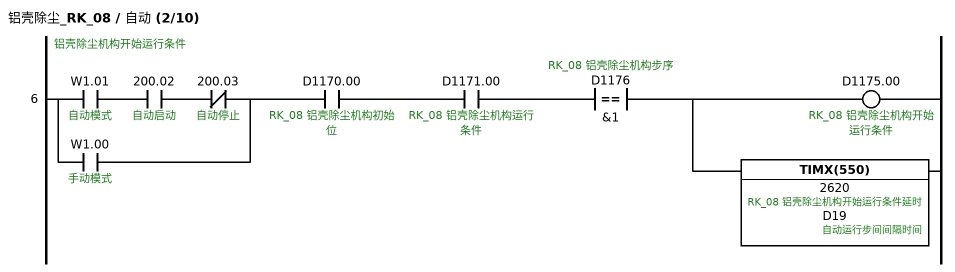
; [picture p624: 铝壳除尘_RK_08 / 自动, rungs 6-6]
; rung 6: 铝壳除尘机构开始运行条件
LD W1.01  ; 自动模式
AND 200.02  ; 自动启动
ANDNOT 200.03  ; 自动停止
OR W1.00  ; 手动模式
AND D1170.00  ; RK_08 铝壳除尘机构初始位
AND D1171.00  ; RK_08 铝壳除尘机构运行条件
AND=(300) D1176 &1  ; RK_08 铝壳除尘机构步序
OUT D1175.00  ; RK_08 铝壳除尘机构开始运行条件
TIMX(550) 2620 D19  ; 自动运行步间间隔时间, RK_08 铝壳除尘机构开始运行条件延时

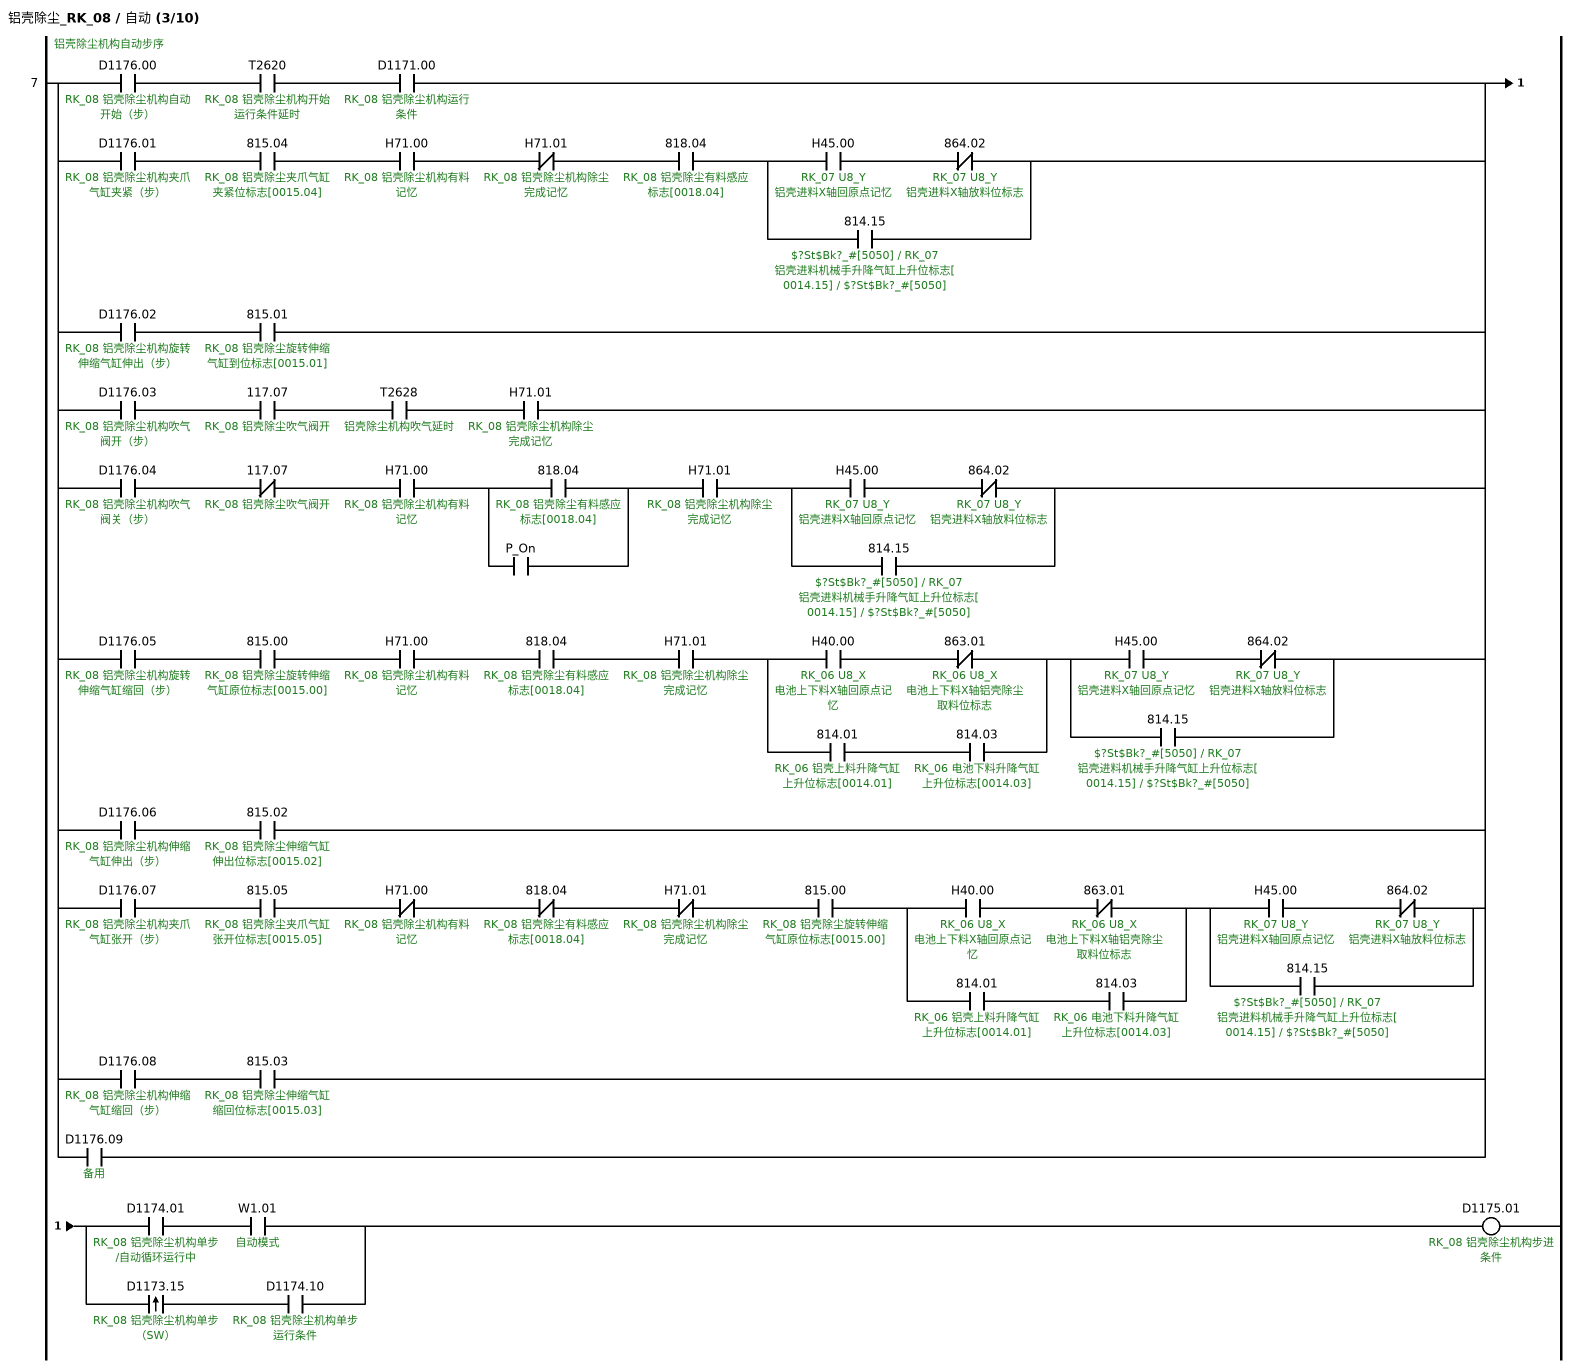
; rung 7: 铝壳除尘机构自动步序
LD D1176.00  ; RK_08 铝壳除尘机构自动开始（步）
AND T2620  ; RK_08 铝壳除尘机构开始运行条件延时
AND D1171.00  ; RK_08 铝壳除尘机构运行条件
LD D1176.01  ; RK_08 铝壳除尘机构夹爪气缸夹紧（步）
AND 815.04  ; RK_08 铝壳除尘夹爪气缸夹紧位标志[0015.04]
AND H71.00  ; RK_08 铝壳除尘机构有料记忆
ANDNOT H71.01  ; RK_08 铝壳除尘机构除尘完成记忆
AND 818.04  ; RK_08 铝壳除尘有料感应标志[0018.04]
LD H45.00  ; RK_07 U8_Y 铝壳进料X轴回原点记忆
ANDNOT 864.02  ; RK_07 U8_Y 铝壳进料X轴放料位标志
OR 814.15  ; $?St$Bk?_#[5050] / RK_07 铝壳进料机械手升降气缸上升位标志[0014.15] / $?St$Bk?_#[5050]
ANDLD
ORLD
LD D1176.02  ; RK_08 铝壳除尘机构旋转伸缩气缸伸出（步）
AND 815.01  ; RK_08 铝壳除尘旋转伸缩气缸到位标志[0015.01]
ORLD
LD D1176.03  ; RK_08 铝壳除尘机构吹气阀开（步）
AND 117.07  ; RK_08 铝壳除尘吹气阀开
AND T2628  ; 铝壳除尘机构吹气延时
AND H71.01  ; RK_08 铝壳除尘机构除尘完成记忆
ORLD
LD D1176.04  ; RK_08 铝壳除尘机构吹气阀关（步）
ANDNOT 117.07  ; RK_08 铝壳除尘吹气阀开
AND H71.00  ; RK_08 铝壳除尘机构有料记忆
LD 818.04  ; RK_08 铝壳除尘有料感应标志[0018.04]
OR P_On
ANDLD
AND H71.01  ; RK_08 铝壳除尘机构除尘完成记忆
LD H45.00  ; RK_07 U8_Y 铝壳进料X轴回原点记忆
ANDNOT 864.02  ; RK_07 U8_Y 铝壳进料X轴放料位标志
OR 814.15  ; $?St$Bk?_#[5050] / RK_07 铝壳进料机械手升降气缸上升位标志[0014.15] / $?St$Bk?_#[5050]
ANDLD
ORLD
LD D1176.05  ; RK_08 铝壳除尘机构旋转伸缩气缸缩回（步）
AND 815.00  ; RK_08 铝壳除尘旋转伸缩气缸原位标志[0015.00]
AND H71.00  ; RK_08 铝壳除尘机构有料记忆
AND 818.04  ; RK_08 铝壳除尘有料感应标志[0018.04]
AND H71.01  ; RK_08 铝壳除尘机构除尘完成记忆
LD H40.00  ; RK_06 U8_X 电池上下料X轴回原点记忆
ANDNOT 863.01  ; RK_06 U8_X 电池上下料X轴铝壳除尘取料位标志
LD 814.01  ; RK_06 铝壳上料升降气缸上升位标志[0014.01]
AND 814.03  ; RK_06 电池下料升降气缸上升位标志[0014.03]
ORLD
ANDLD
LD H45.00  ; RK_07 U8_Y 铝壳进料X轴回原点记忆
ANDNOT 864.02  ; RK_07 U8_Y 铝壳进料X轴放料位标志
OR 814.15  ; $?St$Bk?_#[5050] / RK_07 铝壳进料机械手升降气缸上升位标志[0014.15] / $?St$Bk?_#[5050]
ANDLD
ORLD
LD D1176.06  ; RK_08 铝壳除尘机构伸缩气缸伸出（步）
AND 815.02  ; RK_08 铝壳除尘伸缩气缸伸出位标志[0015.02]
ORLD
LD D1176.07  ; RK_08 铝壳除尘机构夹爪气缸张开（步）
AND 815.05  ; RK_08 铝壳除尘夹爪气缸张开位标志[0015.05]
ANDNOT H71.00  ; RK_08 铝壳除尘机构有料记忆
ANDNOT 818.04  ; RK_08 铝壳除尘有料感应标志[0018.04]
ANDNOT H71.01  ; RK_08 铝壳除尘机构除尘完成记忆
AND 815.00  ; RK_08 铝壳除尘旋转伸缩气缸原位标志[0015.00]
LD H40.00  ; RK_06 U8_X 电池上下料X轴回原点记忆
ANDNOT 863.01  ; RK_06 U8_X 电池上下料X轴铝壳除尘取料位标志
LD 814.01  ; RK_06 铝壳上料升降气缸上升位标志[0014.01]
AND 814.03  ; RK_06 电池下料升降气缸上升位标志[0014.03]
ORLD
ANDLD
LD H45.00  ; RK_07 U8_Y 铝壳进料X轴回原点记忆
ANDNOT 864.02  ; RK_07 U8_Y 铝壳进料X轴放料位标志
OR 814.15  ; $?St$Bk?_#[5050] / RK_07 铝壳进料机械手升降气缸上升位标志[0014.15] / $?St$Bk?_#[5050]
ANDLD
ORLD
LD D1176.08  ; RK_08 铝壳除尘机构伸缩气缸缩回（步）
AND 815.03  ; RK_08 铝壳除尘伸缩气缸缩回位标志[0015.03]
ORLD
OR D1176.09  ; 备用
LD D1174.01  ; RK_08 铝壳除尘机构单步/自动循环运行中
AND W1.01  ; 自动模式
@LD D1173.15  ; RK_08 铝壳除尘机构单步（SW）
AND D1174.10  ; RK_08 铝壳除尘机构单步运行条件
ORLD
ANDLD
OUT D1175.01  ; RK_08 铝壳除尘机构步进条件

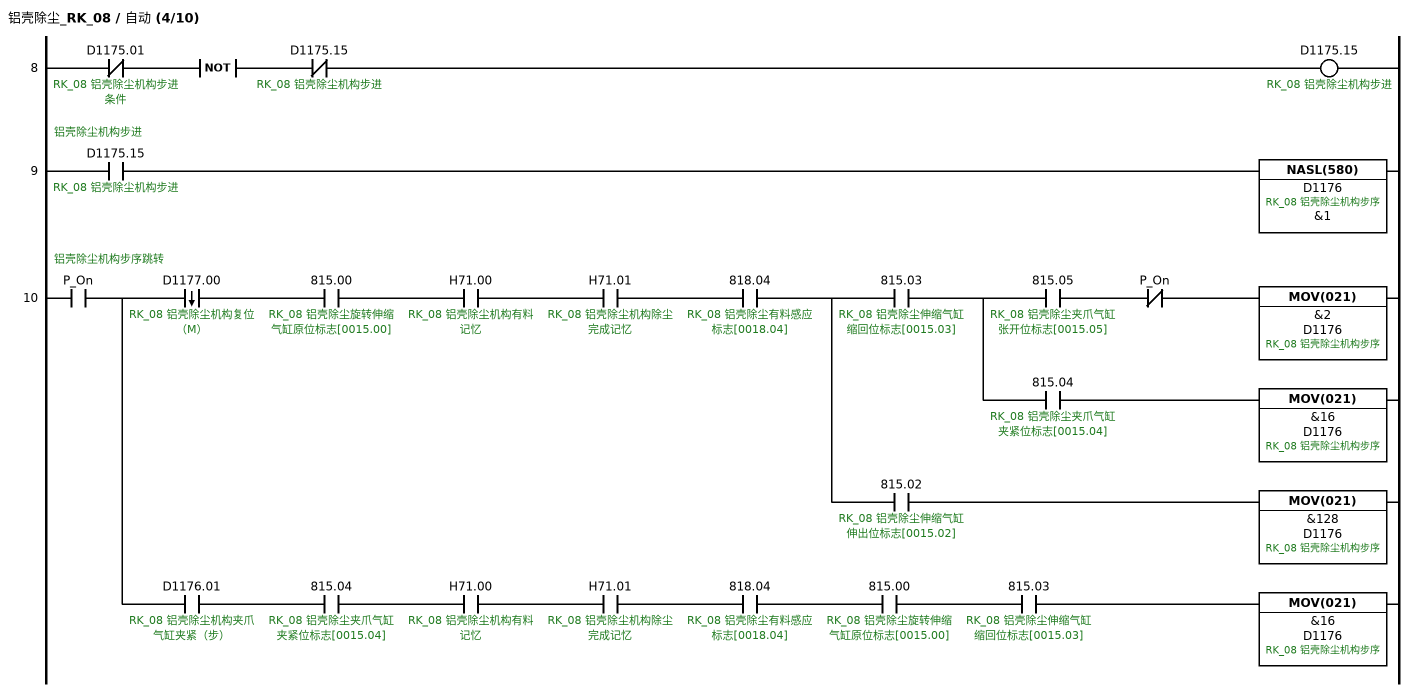
; rung 8
LDNOT D1175.01  ; RK_08 铝壳除尘机构步进条件
NOT(520)
ANDNOT D1175.15  ; RK_08 铝壳除尘机构步进
OUT D1175.15  ; RK_08 铝壳除尘机构步进
; rung 9: 铝壳除尘机构步进
LD D1175.15  ; RK_08 铝壳除尘机构步进
NASL(580) D1176 &1  ; RK_08 铝壳除尘机构步序
; rung 10: 铝壳除尘机构步序跳转
LD P_On
OUT TR0
%AND D1177.00  ; RK_08 铝壳除尘机构复位（M）
AND 815.00  ; RK_08 铝壳除尘旋转伸缩气缸原位标志[0015.00]
AND H71.00  ; RK_08 铝壳除尘机构有料记忆
AND H71.01  ; RK_08 铝壳除尘机构除尘完成记忆
AND 818.04  ; RK_08 铝壳除尘有料感应标志[0018.04]
OUT TR1
AND 815.03  ; RK_08 铝壳除尘伸缩气缸缩回位标志[0015.03]
OUT TR2
AND 815.05  ; RK_08 铝壳除尘夹爪气缸张开位标志[0015.05]
ANDNOT P_On
MOV(021) &2 D1176  ; RK_08 铝壳除尘机构步序  // RK_08 铝壳除尘机构夹爪气缸夹紧步（D1176.01）
LD TR2
AND 815.04  ; RK_08 铝壳除尘夹爪气缸夹紧位标志[0015.04]
MOV(021) &16 D1176  ; RK_08 铝壳除尘机构步序  // RK_08 铝壳除尘机构吹气阀关步（D1176.04）
LD TR1
AND 815.02  ; RK_08 铝壳除尘伸缩气缸伸出位标志[0015.02]
MOV(021) &128 D1176  ; RK_08 铝壳除尘机构步序  // RK_08 铝壳除尘机构夹爪气缸张开步（D1176.07）
LD TR0
AND D1176.01  ; RK_08 铝壳除尘机构夹爪气缸夹紧（步）
AND 815.04  ; RK_08 铝壳除尘夹爪气缸夹紧位标志[0015.04]
AND H71.00  ; RK_08 铝壳除尘机构有料记忆
AND H71.01  ; RK_08 铝壳除尘机构除尘完成记忆
AND 818.04  ; RK_08 铝壳除尘有料感应标志[0018.04]
AND 815.00  ; RK_08 铝壳除尘旋转伸缩气缸原位标志[0015.00]
AND 815.03  ; RK_08 铝壳除尘伸缩气缸缩回位标志[0015.03]
MOV(021) &16 D1176  ; RK_08 铝壳除尘机构步序  // RK_08 铝壳除尘机构吹气阀关步（D1176.04）

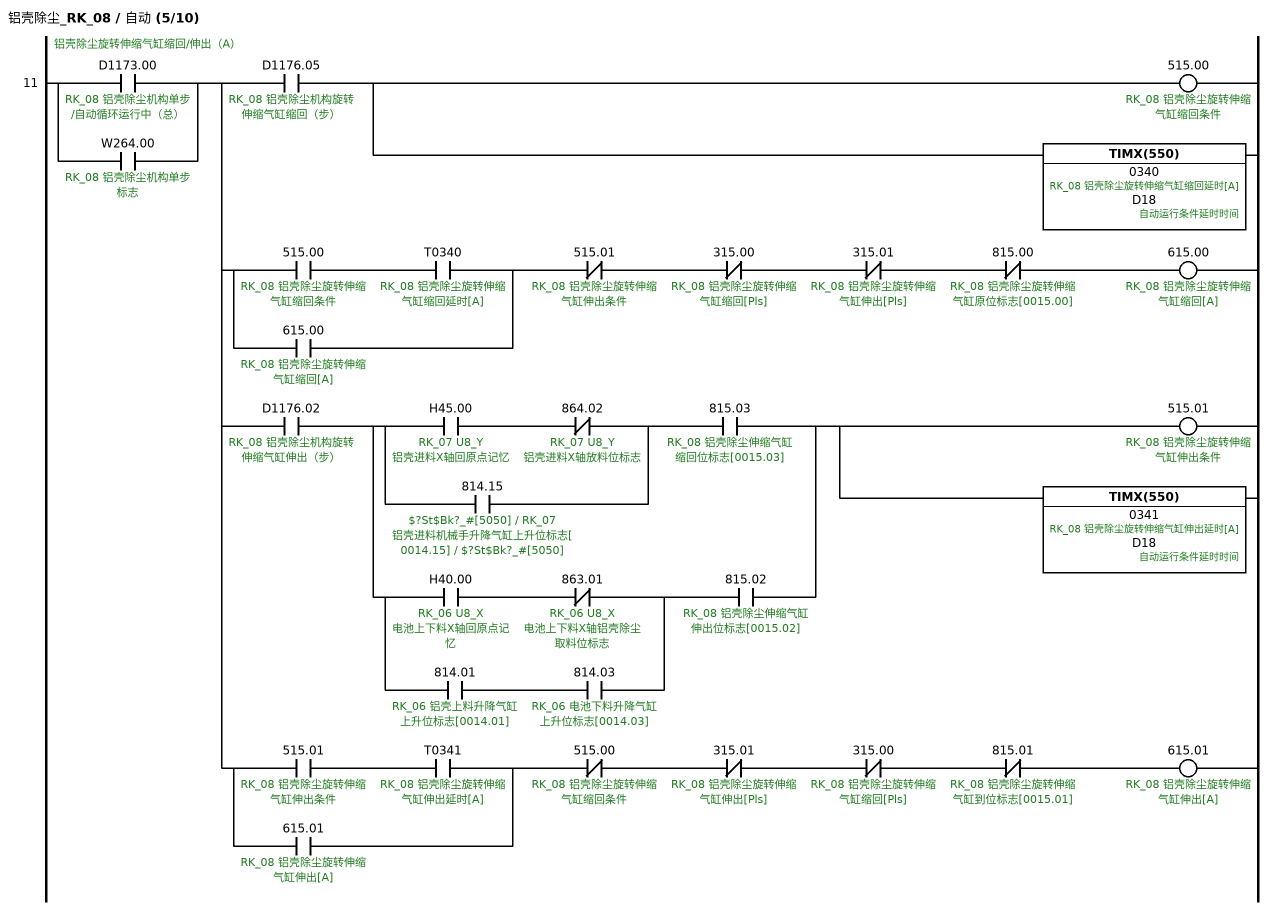
; rung 11: 铝壳除尘旋转伸缩气缸缩回/伸出（A）
LD D1173.00  ; RK_08 铝壳除尘机构单步/自动循环运行中（总）
OR W264.00  ; RK_08 铝壳除尘机构单步标志
OUT TR0
AND D1176.05  ; RK_08 铝壳除尘机构旋转伸缩气缸缩回（步）
OUT 515.00  ; RK_08 铝壳除尘旋转伸缩气缸缩回条件
TIMX(550) 0340 D18  ; 自动运行条件延时时间, RK_08 铝壳除尘旋转伸缩气缸缩回延时[A]
LD TR0
LD 515.00  ; RK_08 铝壳除尘旋转伸缩气缸缩回条件
AND T0340  ; RK_08 铝壳除尘旋转伸缩气缸缩回延时[A]
OR 615.00  ; RK_08 铝壳除尘旋转伸缩气缸缩回[A]
ANDLD
ANDNOT 515.01  ; RK_08 铝壳除尘旋转伸缩气缸伸出条件
ANDNOT 315.00  ; RK_08 铝壳除尘旋转伸缩气缸缩回[Pls]
ANDNOT 315.01  ; RK_08 铝壳除尘旋转伸缩气缸伸出[Pls]
ANDNOT 815.00  ; RK_08 铝壳除尘旋转伸缩气缸原位标志[0015.00]
OUT 615.00  ; RK_08 铝壳除尘旋转伸缩气缸缩回[A]
LD TR0
AND D1176.02  ; RK_08 铝壳除尘机构旋转伸缩气缸伸出（步）
LD H45.00  ; RK_07 U8_Y 铝壳进料X轴回原点记忆
ANDNOT 864.02  ; RK_07 U8_Y 铝壳进料X轴放料位标志
OR 814.15  ; $?St$Bk?_#[5050] / RK_07 铝壳进料机械手升降气缸上升位标志[0014.15] / $?St$Bk?_#[5050]
AND 815.03  ; RK_08 铝壳除尘伸缩气缸缩回位标志[0015.03]
LD H40.00  ; RK_06 U8_X 电池上下料X轴回原点记忆
ANDNOT 863.01  ; RK_06 U8_X 电池上下料X轴铝壳除尘取料位标志
LD 814.01  ; RK_06 铝壳上料升降气缸上升位标志[0014.01]
AND 814.03  ; RK_06 电池下料升降气缸上升位标志[0014.03]
ORLD
AND 815.02  ; RK_08 铝壳除尘伸缩气缸伸出位标志[0015.02]
ORLD
ANDLD
OUT 515.01  ; RK_08 铝壳除尘旋转伸缩气缸伸出条件
TIMX(550) 0341 D18  ; 自动运行条件延时时间, RK_08 铝壳除尘旋转伸缩气缸伸出延时[A]
LD TR0
LD 515.01  ; RK_08 铝壳除尘旋转伸缩气缸伸出条件
AND T0341  ; RK_08 铝壳除尘旋转伸缩气缸伸出延时[A]
OR 615.01  ; RK_08 铝壳除尘旋转伸缩气缸伸出[A]
ANDLD
ANDNOT 515.00  ; RK_08 铝壳除尘旋转伸缩气缸缩回条件
ANDNOT 315.01  ; RK_08 铝壳除尘旋转伸缩气缸伸出[Pls]
ANDNOT 315.00  ; RK_08 铝壳除尘旋转伸缩气缸缩回[Pls]
ANDNOT 815.01  ; RK_08 铝壳除尘旋转伸缩气缸到位标志[0015.01]
OUT 615.01  ; RK_08 铝壳除尘旋转伸缩气缸伸出[A]

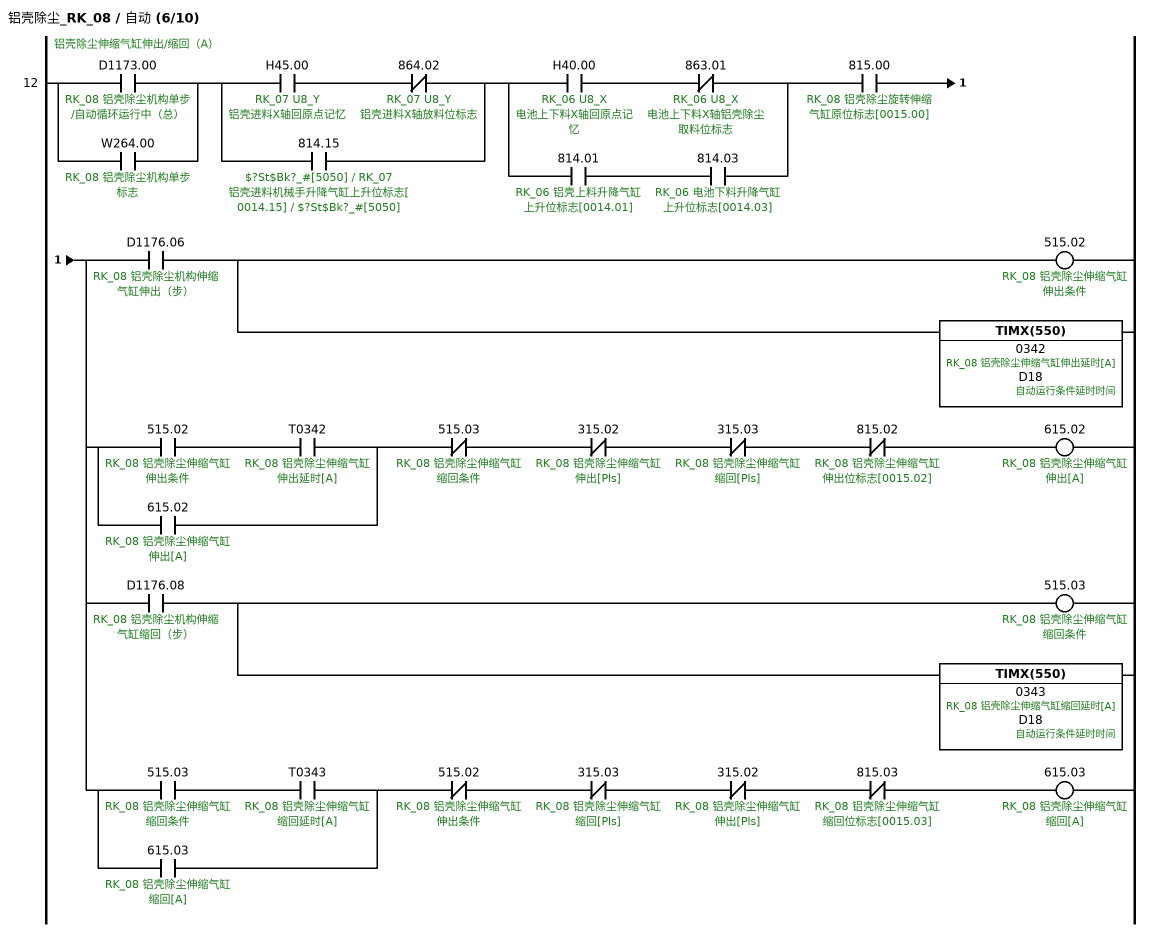
; rung 12: 铝壳除尘伸缩气缸伸出/缩回（A）
LD D1173.00  ; RK_08 铝壳除尘机构单步/自动循环运行中（总）
OR W264.00  ; RK_08 铝壳除尘机构单步标志
LD H45.00  ; RK_07 U8_Y 铝壳进料X轴回原点记忆
ANDNOT 864.02  ; RK_07 U8_Y 铝壳进料X轴放料位标志
OR 814.15  ; $?St$Bk?_#[5050] / RK_07 铝壳进料机械手升降气缸上升位标志[0014.15] / $?St$Bk?_#[5050]
ANDLD
LD H40.00  ; RK_06 U8_X 电池上下料X轴回原点记忆
ANDNOT 863.01  ; RK_06 U8_X 电池上下料X轴铝壳除尘取料位标志
LD 814.01  ; RK_06 铝壳上料升降气缸上升位标志[0014.01]
AND 814.03  ; RK_06 电池下料升降气缸上升位标志[0014.03]
ORLD
ANDLD
AND 815.00  ; RK_08 铝壳除尘旋转伸缩气缸原位标志[0015.00]
OUT TR0
AND D1176.06  ; RK_08 铝壳除尘机构伸缩气缸伸出（步）
OUT 515.02  ; RK_08 铝壳除尘伸缩气缸伸出条件
TIMX(550) 0342 D18  ; 自动运行条件延时时间, RK_08 铝壳除尘伸缩气缸伸出延时[A]
LD TR0
LD 515.02  ; RK_08 铝壳除尘伸缩气缸伸出条件
AND T0342  ; RK_08 铝壳除尘伸缩气缸伸出延时[A]
OR 615.02  ; RK_08 铝壳除尘伸缩气缸伸出[A]
ANDLD
ANDNOT 515.03  ; RK_08 铝壳除尘伸缩气缸缩回条件
ANDNOT 315.02  ; RK_08 铝壳除尘伸缩气缸伸出[Pls]
ANDNOT 315.03  ; RK_08 铝壳除尘伸缩气缸缩回[Pls]
ANDNOT 815.02  ; RK_08 铝壳除尘伸缩气缸伸出位标志[0015.02]
OUT 615.02  ; RK_08 铝壳除尘伸缩气缸伸出[A]
LD TR0
AND D1176.08  ; RK_08 铝壳除尘机构伸缩气缸缩回（步）
OUT 515.03  ; RK_08 铝壳除尘伸缩气缸缩回条件
TIMX(550) 0343 D18  ; 自动运行条件延时时间, RK_08 铝壳除尘伸缩气缸缩回延时[A]
LD TR0
LD 515.03  ; RK_08 铝壳除尘伸缩气缸缩回条件
AND T0343  ; RK_08 铝壳除尘伸缩气缸缩回延时[A]
OR 615.03  ; RK_08 铝壳除尘伸缩气缸缩回[A]
ANDLD
ANDNOT 515.02  ; RK_08 铝壳除尘伸缩气缸伸出条件
ANDNOT 315.03  ; RK_08 铝壳除尘伸缩气缸缩回[Pls]
ANDNOT 315.02  ; RK_08 铝壳除尘伸缩气缸伸出[Pls]
ANDNOT 815.03  ; RK_08 铝壳除尘伸缩气缸缩回位标志[0015.03]
OUT 615.03  ; RK_08 铝壳除尘伸缩气缸缩回[A]

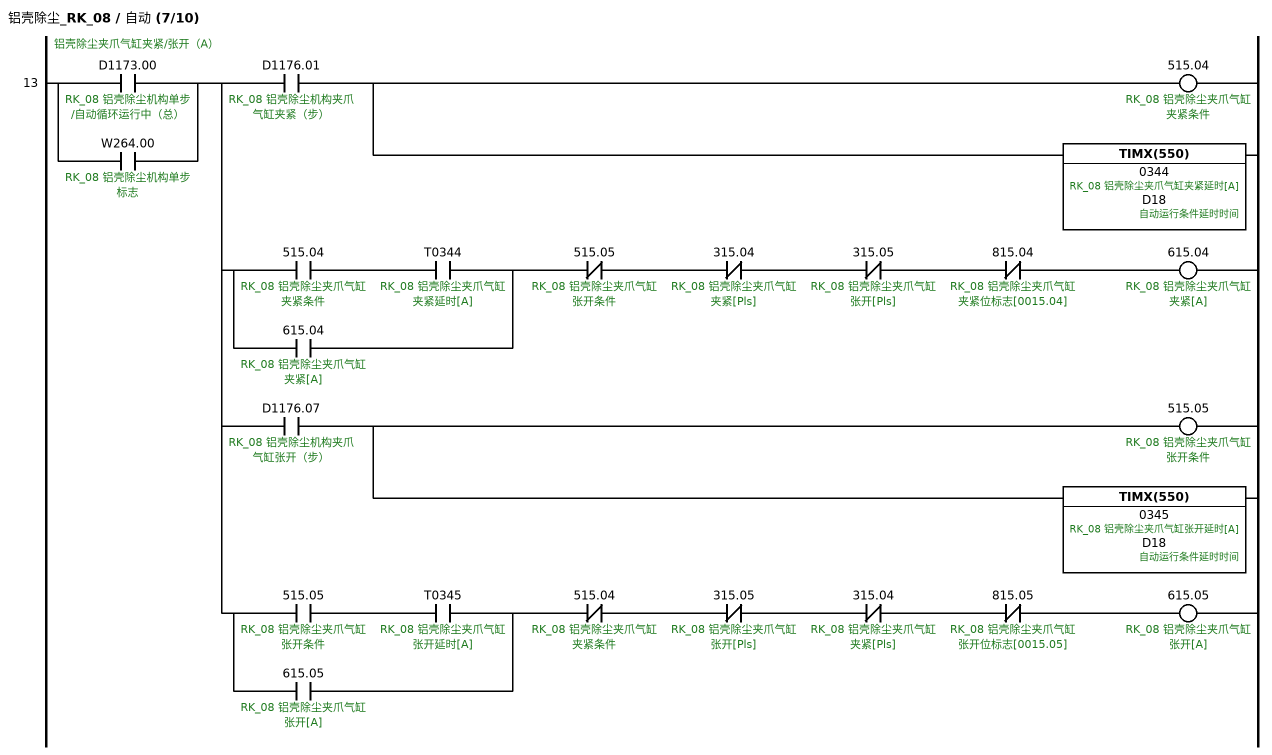
; rung 13: 铝壳除尘夹爪气缸夹紧/张开（A）
LD D1173.00  ; RK_08 铝壳除尘机构单步/自动循环运行中（总）
OR W264.00  ; RK_08 铝壳除尘机构单步标志
OUT TR0
AND D1176.01  ; RK_08 铝壳除尘机构夹爪气缸夹紧（步）
OUT 515.04  ; RK_08 铝壳除尘夹爪气缸夹紧条件
TIMX(550) 0344 D18  ; 自动运行条件延时时间, RK_08 铝壳除尘夹爪气缸夹紧延时[A]
LD TR0
LD 515.04  ; RK_08 铝壳除尘夹爪气缸夹紧条件
AND T0344  ; RK_08 铝壳除尘夹爪气缸夹紧延时[A]
OR 615.04  ; RK_08 铝壳除尘夹爪气缸夹紧[A]
ANDLD
ANDNOT 515.05  ; RK_08 铝壳除尘夹爪气缸张开条件
ANDNOT 315.04  ; RK_08 铝壳除尘夹爪气缸夹紧[Pls]
ANDNOT 315.05  ; RK_08 铝壳除尘夹爪气缸张开[Pls]
ANDNOT 815.04  ; RK_08 铝壳除尘夹爪气缸夹紧位标志[0015.04]
OUT 615.04  ; RK_08 铝壳除尘夹爪气缸夹紧[A]
LD TR0
AND D1176.07  ; RK_08 铝壳除尘机构夹爪气缸张开（步）
OUT 515.05  ; RK_08 铝壳除尘夹爪气缸张开条件
TIMX(550) 0345 D18  ; 自动运行条件延时时间, RK_08 铝壳除尘夹爪气缸张开延时[A]
LD TR0
LD 515.05  ; RK_08 铝壳除尘夹爪气缸张开条件
AND T0345  ; RK_08 铝壳除尘夹爪气缸张开延时[A]
OR 615.05  ; RK_08 铝壳除尘夹爪气缸张开[A]
ANDLD
ANDNOT 515.04  ; RK_08 铝壳除尘夹爪气缸夹紧条件
ANDNOT 315.05  ; RK_08 铝壳除尘夹爪气缸张开[Pls]
ANDNOT 315.04  ; RK_08 铝壳除尘夹爪气缸夹紧[Pls]
ANDNOT 815.05  ; RK_08 铝壳除尘夹爪气缸张开位标志[0015.05]
OUT 615.05  ; RK_08 铝壳除尘夹爪气缸张开[A]

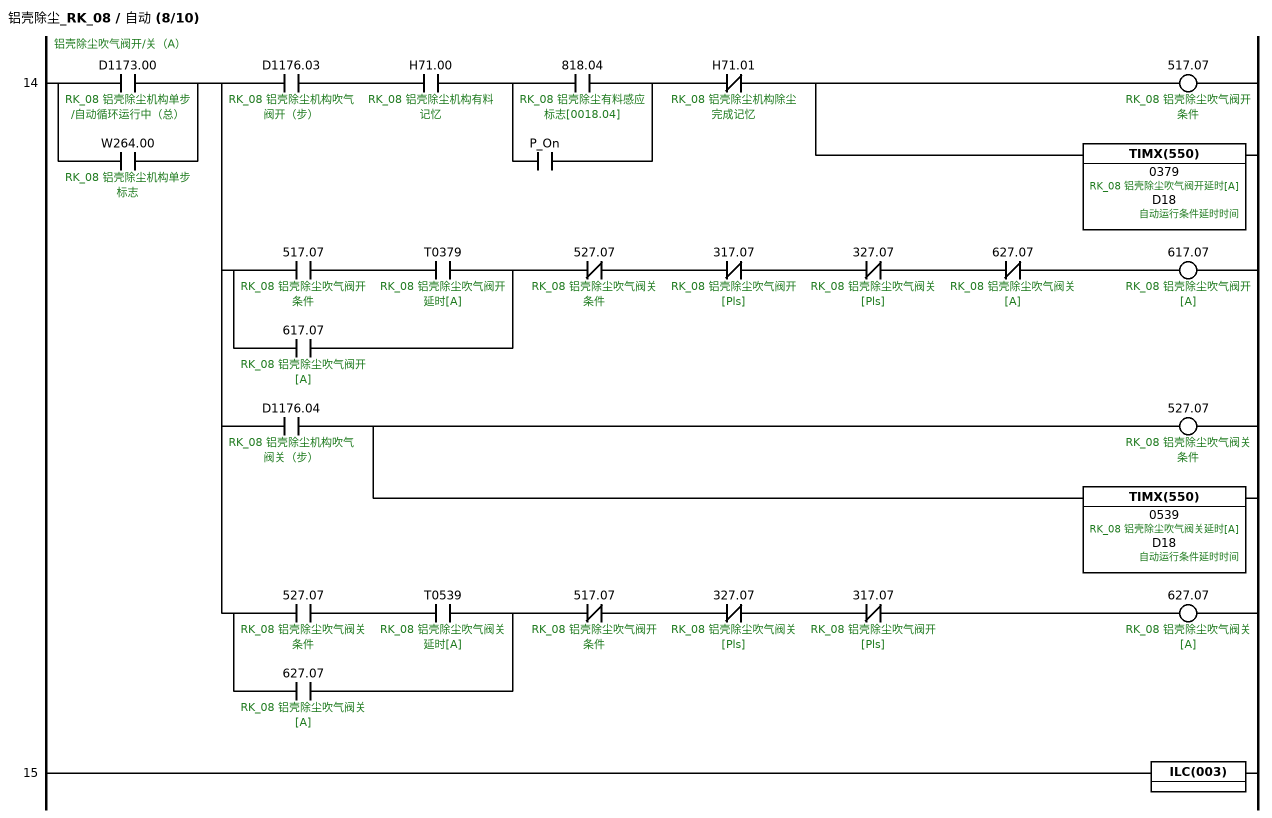
; rung 14: 铝壳除尘吹气阀开/关（A）
LD D1173.00  ; RK_08 铝壳除尘机构单步/自动循环运行中（总）
OR W264.00  ; RK_08 铝壳除尘机构单步标志
OUT TR0
AND D1176.03  ; RK_08 铝壳除尘机构吹气阀开（步）
AND H71.00  ; RK_08 铝壳除尘机构有料记忆
LD 818.04  ; RK_08 铝壳除尘有料感应标志[0018.04]
OR P_On
ANDLD
ANDNOT H71.01  ; RK_08 铝壳除尘机构除尘完成记忆
OUT 517.07  ; RK_08 铝壳除尘吹气阀开条件
TIMX(550) 0379 D18  ; 自动运行条件延时时间, RK_08 铝壳除尘吹气阀开延时[A]
LD TR0
LD 517.07  ; RK_08 铝壳除尘吹气阀开条件
AND T0379  ; RK_08 铝壳除尘吹气阀开延时[A]
OR 617.07  ; RK_08 铝壳除尘吹气阀开[A]
ANDLD
ANDNOT 527.07  ; RK_08 铝壳除尘吹气阀关条件
ANDNOT 317.07  ; RK_08 铝壳除尘吹气阀开[Pls]
ANDNOT 327.07  ; RK_08 铝壳除尘吹气阀关[Pls]
ANDNOT 627.07  ; RK_08 铝壳除尘吹气阀关[A]
OUT 617.07  ; RK_08 铝壳除尘吹气阀开[A]
LD TR0
AND D1176.04  ; RK_08 铝壳除尘机构吹气阀关（步）
OUT 527.07  ; RK_08 铝壳除尘吹气阀关条件
TIMX(550) 0539 D18  ; 自动运行条件延时时间, RK_08 铝壳除尘吹气阀关延时[A]
LD TR0
LD 527.07  ; RK_08 铝壳除尘吹气阀关条件
AND T0539  ; RK_08 铝壳除尘吹气阀关延时[A]
OR 627.07  ; RK_08 铝壳除尘吹气阀关[A]
ANDLD
ANDNOT 517.07  ; RK_08 铝壳除尘吹气阀开条件
ANDNOT 327.07  ; RK_08 铝壳除尘吹气阀关[Pls]
ANDNOT 317.07  ; RK_08 铝壳除尘吹气阀开[Pls]
OUT 627.07  ; RK_08 铝壳除尘吹气阀关[A]
; rung 15
ILC(003)

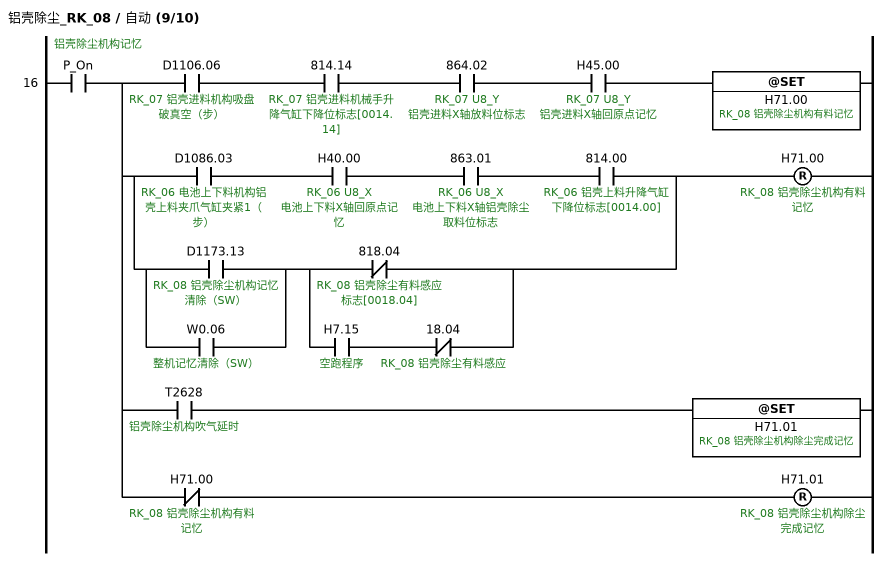
; rung 16: 铝壳除尘机构记忆
LD P_On
OUT TR0
AND D1106.06  ; RK_07 铝壳进料机构吸盘破真空（步）
AND 814.14  ; RK_07 铝壳进料机械手升降气缸下降位标志[0014.14]
AND 864.02  ; RK_07 U8_Y 铝壳进料X轴放料位标志
AND H45.00  ; RK_07 U8_Y 铝壳进料X轴回原点记忆
@SET H71.00  ; RK_08 铝壳除尘机构有料记忆
LD TR0
LD D1086.03  ; RK_06 电池上下料机构铝壳上料夹爪气缸夹紧1（步）
AND H40.00  ; RK_06 U8_X 电池上下料X轴回原点记忆
AND 863.01  ; RK_06 U8_X 电池上下料X轴铝壳除尘取料位标志
AND 814.00  ; RK_06 铝壳上料升降气缸下降位标志[0014.00]
LD D1173.13  ; RK_08 铝壳除尘机构记忆清除（SW）
OR W0.06  ; 整机记忆清除（SW）
LDNOT 818.04  ; RK_08 铝壳除尘有料感应标志[0018.04]
LD H7.15  ; 空跑程序
ANDNOT 18.04  ; RK_08 铝壳除尘有料感应
ORLD
ANDLD
ORLD
ANDLD
RSET H71.00  ; RK_08 铝壳除尘机构有料记忆
LD TR0
AND T2628  ; 铝壳除尘机构吹气延时
@SET H71.01  ; RK_08 铝壳除尘机构除尘完成记忆
LD TR0
ANDNOT H71.00  ; RK_08 铝壳除尘机构有料记忆
RSET H71.01  ; RK_08 铝壳除尘机构除尘完成记忆

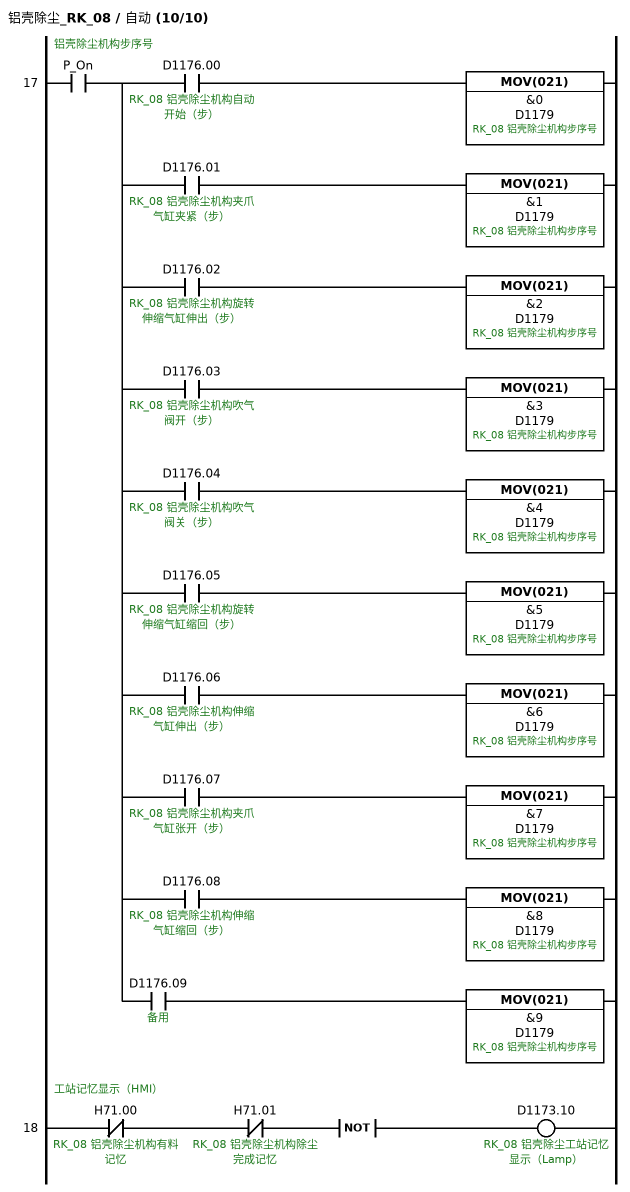
; rung 17: 铝壳除尘机构步序号
LD P_On
OUT TR0
AND D1176.00  ; RK_08 铝壳除尘机构自动开始（步）
MOV(021) &0 D1179  ; RK_08 铝壳除尘机构步序号
LD TR0
AND D1176.01  ; RK_08 铝壳除尘机构夹爪气缸夹紧（步）
MOV(021) &1 D1179  ; RK_08 铝壳除尘机构步序号
LD TR0
AND D1176.02  ; RK_08 铝壳除尘机构旋转伸缩气缸伸出（步）
MOV(021) &2 D1179  ; RK_08 铝壳除尘机构步序号
LD TR0
AND D1176.03  ; RK_08 铝壳除尘机构吹气阀开（步）
MOV(021) &3 D1179  ; RK_08 铝壳除尘机构步序号
LD TR0
AND D1176.04  ; RK_08 铝壳除尘机构吹气阀关（步）
MOV(021) &4 D1179  ; RK_08 铝壳除尘机构步序号
LD TR0
AND D1176.05  ; RK_08 铝壳除尘机构旋转伸缩气缸缩回（步）
MOV(021) &5 D1179  ; RK_08 铝壳除尘机构步序号
LD TR0
AND D1176.06  ; RK_08 铝壳除尘机构伸缩气缸伸出（步）
MOV(021) &6 D1179  ; RK_08 铝壳除尘机构步序号
LD TR0
AND D1176.07  ; RK_08 铝壳除尘机构夹爪气缸张开（步）
MOV(021) &7 D1179  ; RK_08 铝壳除尘机构步序号
LD TR0
AND D1176.08  ; RK_08 铝壳除尘机构伸缩气缸缩回（步）
MOV(021) &8 D1179  ; RK_08 铝壳除尘机构步序号
LD TR0
AND D1176.09  ; 备用
MOV(021) &9 D1179  ; RK_08 铝壳除尘机构步序号
; rung 18: 工站记忆显示（HMI）
LDNOT H71.00  ; RK_08 铝壳除尘机构有料记忆
ANDNOT H71.01  ; RK_08 铝壳除尘机构除尘完成记忆
NOT(520)
OUT D1173.10  ; RK_08 铝壳除尘工站记忆显示（Lamp）

### Section 复位

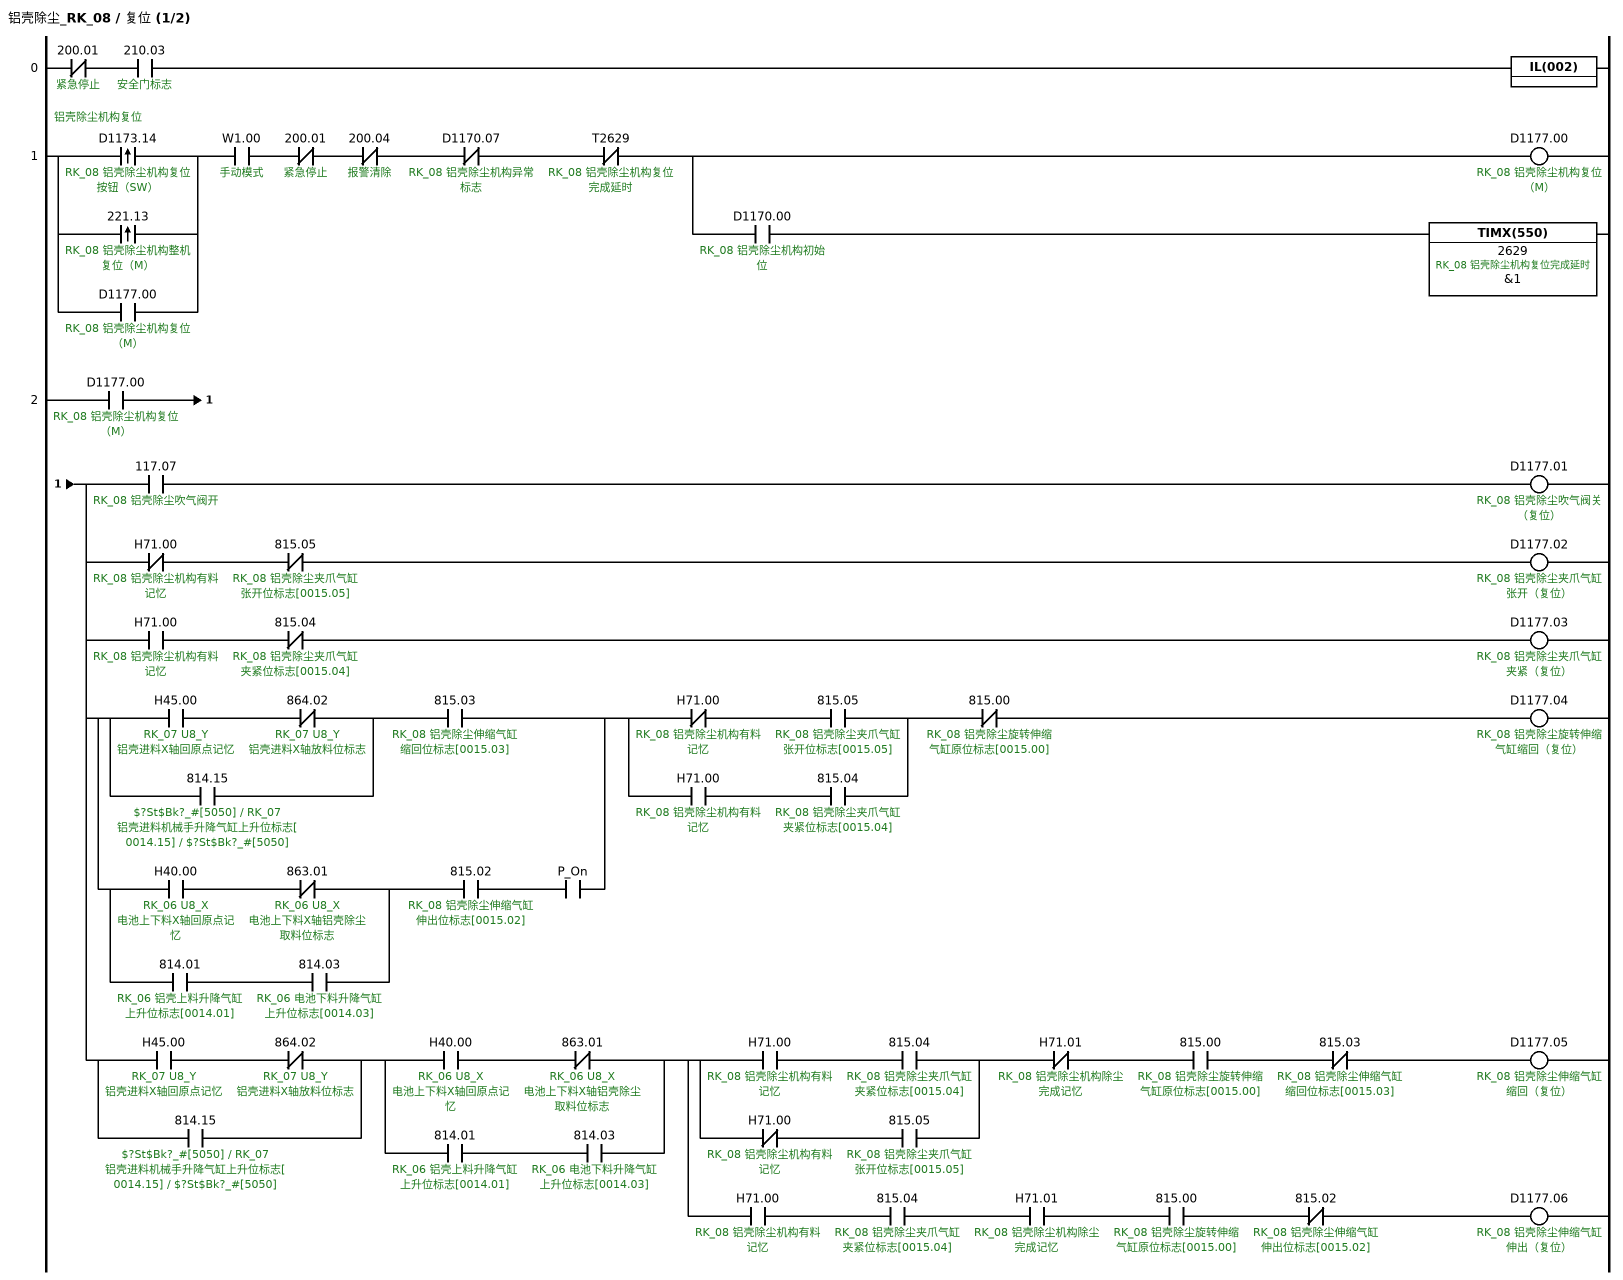
; rung 0
LDNOT 200.01  ; 紧急停止
AND 210.03  ; 安全门标志
IL(002)
; rung 1: 铝壳除尘机构复位
@LD D1173.14  ; RK_08 铝壳除尘机构复位按钮（SW）
@OR 221.13  ; RK_08 铝壳除尘机构整机复位（M）
OR D1177.00  ; RK_08 铝壳除尘机构复位（M）
AND W1.00  ; 手动模式
ANDNOT 200.01  ; 紧急停止
ANDNOT 200.04  ; 报警清除
ANDNOT D1170.07  ; RK_08 铝壳除尘机构异常标志
ANDNOT T2629  ; RK_08 铝壳除尘机构复位完成延时
OUT D1177.00  ; RK_08 铝壳除尘机构复位（M）
AND D1170.00  ; RK_08 铝壳除尘机构初始位
TIMX(550) 2629 &1  ; RK_08 铝壳除尘机构复位完成延时
; rung 2
LD D1177.00  ; RK_08 铝壳除尘机构复位（M）
OUT TR0
AND 117.07  ; RK_08 铝壳除尘吹气阀开
OUT D1177.01  ; RK_08 铝壳除尘吹气阀关（复位）
LD TR0
ANDNOT H71.00  ; RK_08 铝壳除尘机构有料记忆
ANDNOT 815.05  ; RK_08 铝壳除尘夹爪气缸张开位标志[0015.05]
OUT D1177.02  ; RK_08 铝壳除尘夹爪气缸张开（复位）
LD TR0
AND H71.00  ; RK_08 铝壳除尘机构有料记忆
ANDNOT 815.04  ; RK_08 铝壳除尘夹爪气缸夹紧位标志[0015.04]
OUT D1177.03  ; RK_08 铝壳除尘夹爪气缸夹紧（复位）
LD TR0
LD H45.00  ; RK_07 U8_Y 铝壳进料X轴回原点记忆
ANDNOT 864.02  ; RK_07 U8_Y 铝壳进料X轴放料位标志
OR 814.15  ; $?St$Bk?_#[5050] / RK_07 铝壳进料机械手升降气缸上升位标志[0014.15] / $?St$Bk?_#[5050]
AND 815.03  ; RK_08 铝壳除尘伸缩气缸缩回位标志[0015.03]
LD H40.00  ; RK_06 U8_X 电池上下料X轴回原点记忆
ANDNOT 863.01  ; RK_06 U8_X 电池上下料X轴铝壳除尘取料位标志
LD 814.01  ; RK_06 铝壳上料升降气缸上升位标志[0014.01]
AND 814.03  ; RK_06 电池下料升降气缸上升位标志[0014.03]
ORLD
AND 815.02  ; RK_08 铝壳除尘伸缩气缸伸出位标志[0015.02]
AND P_On
ORLD
ANDLD
LDNOT H71.00  ; RK_08 铝壳除尘机构有料记忆
AND 815.05  ; RK_08 铝壳除尘夹爪气缸张开位标志[0015.05]
LD H71.00  ; RK_08 铝壳除尘机构有料记忆
AND 815.04  ; RK_08 铝壳除尘夹爪气缸夹紧位标志[0015.04]
ORLD
ANDLD
ANDNOT 815.00  ; RK_08 铝壳除尘旋转伸缩气缸原位标志[0015.00]
OUT D1177.04  ; RK_08 铝壳除尘旋转伸缩气缸缩回（复位）
LD TR0
LD H45.00  ; RK_07 U8_Y 铝壳进料X轴回原点记忆
ANDNOT 864.02  ; RK_07 U8_Y 铝壳进料X轴放料位标志
OR 814.15  ; $?St$Bk?_#[5050] / RK_07 铝壳进料机械手升降气缸上升位标志[0014.15] / $?St$Bk?_#[5050]
ANDLD
LD H40.00  ; RK_06 U8_X 电池上下料X轴回原点记忆
ANDNOT 863.01  ; RK_06 U8_X 电池上下料X轴铝壳除尘取料位标志
LD 814.01  ; RK_06 铝壳上料升降气缸上升位标志[0014.01]
AND 814.03  ; RK_06 电池下料升降气缸上升位标志[0014.03]
ORLD
ANDLD
OUT TR0
LD H71.00  ; RK_08 铝壳除尘机构有料记忆
AND 815.04  ; RK_08 铝壳除尘夹爪气缸夹紧位标志[0015.04]
LDNOT H71.00  ; RK_08 铝壳除尘机构有料记忆
AND 815.05  ; RK_08 铝壳除尘夹爪气缸张开位标志[0015.05]
ORLD
ANDLD
ANDNOT H71.01  ; RK_08 铝壳除尘机构除尘完成记忆
AND 815.00  ; RK_08 铝壳除尘旋转伸缩气缸原位标志[0015.00]
ANDNOT 815.03  ; RK_08 铝壳除尘伸缩气缸缩回位标志[0015.03]
OUT D1177.05  ; RK_08 铝壳除尘伸缩气缸缩回（复位）
LD TR0
AND H71.00  ; RK_08 铝壳除尘机构有料记忆
AND 815.04  ; RK_08 铝壳除尘夹爪气缸夹紧位标志[0015.04]
AND H71.01  ; RK_08 铝壳除尘机构除尘完成记忆
AND 815.00  ; RK_08 铝壳除尘旋转伸缩气缸原位标志[0015.00]
ANDNOT 815.02  ; RK_08 铝壳除尘伸缩气缸伸出位标志[0015.02]
OUT D1177.06  ; RK_08 铝壳除尘伸缩气缸伸出（复位）

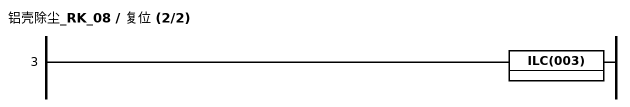
; rung 3
ILC(003)

### Section 指示灯

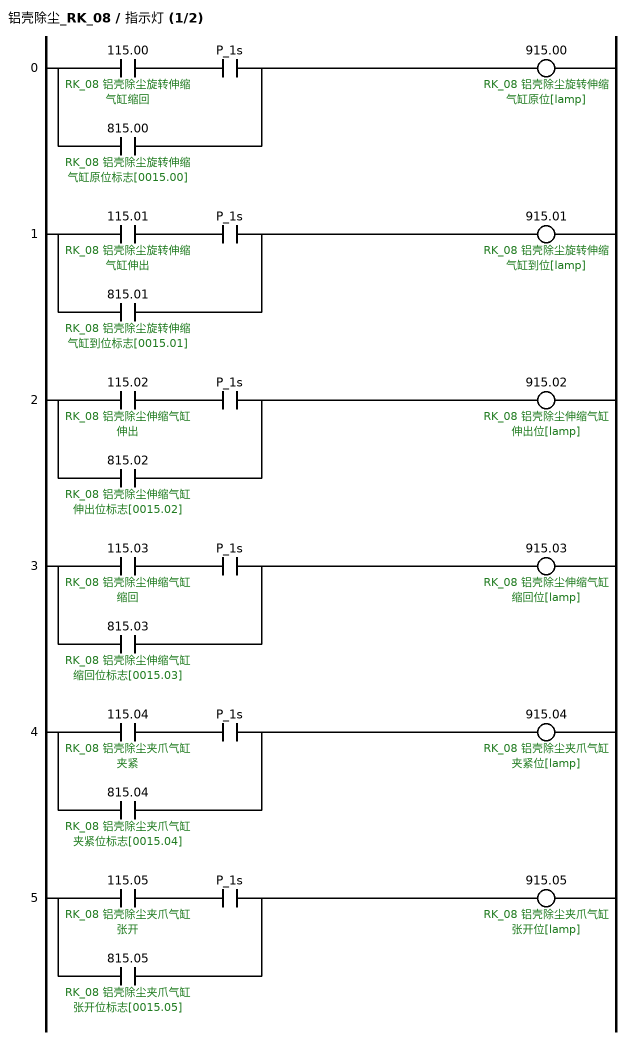
; rung 0
LD 115.00  ; RK_08 铝壳除尘旋转伸缩气缸缩回
AND P_1s
OR 815.00  ; RK_08 铝壳除尘旋转伸缩气缸原位标志[0015.00]
OUT 915.00  ; RK_08 铝壳除尘旋转伸缩气缸原位[lamp]
; rung 1
LD 115.01  ; RK_08 铝壳除尘旋转伸缩气缸伸出
AND P_1s
OR 815.01  ; RK_08 铝壳除尘旋转伸缩气缸到位标志[0015.01]
OUT 915.01  ; RK_08 铝壳除尘旋转伸缩气缸到位[lamp]
; rung 2
LD 115.02  ; RK_08 铝壳除尘伸缩气缸伸出
AND P_1s
OR 815.02  ; RK_08 铝壳除尘伸缩气缸伸出位标志[0015.02]
OUT 915.02  ; RK_08 铝壳除尘伸缩气缸伸出位[lamp]
; rung 3
LD 115.03  ; RK_08 铝壳除尘伸缩气缸缩回
AND P_1s
OR 815.03  ; RK_08 铝壳除尘伸缩气缸缩回位标志[0015.03]
OUT 915.03  ; RK_08 铝壳除尘伸缩气缸缩回位[lamp]
; rung 4
LD 115.04  ; RK_08 铝壳除尘夹爪气缸夹紧
AND P_1s
OR 815.04  ; RK_08 铝壳除尘夹爪气缸夹紧位标志[0015.04]
OUT 915.04  ; RK_08 铝壳除尘夹爪气缸夹紧位[lamp]
; rung 5
LD 115.05  ; RK_08 铝壳除尘夹爪气缸张开
AND P_1s
OR 815.05  ; RK_08 铝壳除尘夹爪气缸张开位标志[0015.05]
OUT 915.05  ; RK_08 铝壳除尘夹爪气缸张开位[lamp]

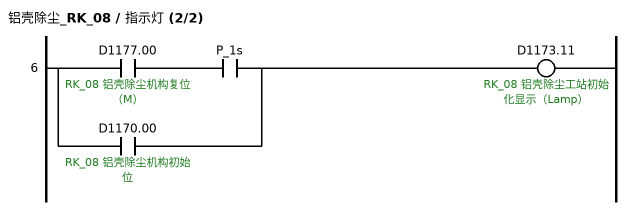
; rung 6
LD D1177.00  ; RK_08 铝壳除尘机构复位（M）
AND P_1s
OR D1170.00  ; RK_08 铝壳除尘机构初始位
OUT D1173.11  ; RK_08 铝壳除尘工站初始化显示（Lamp）

### Section 外部输出

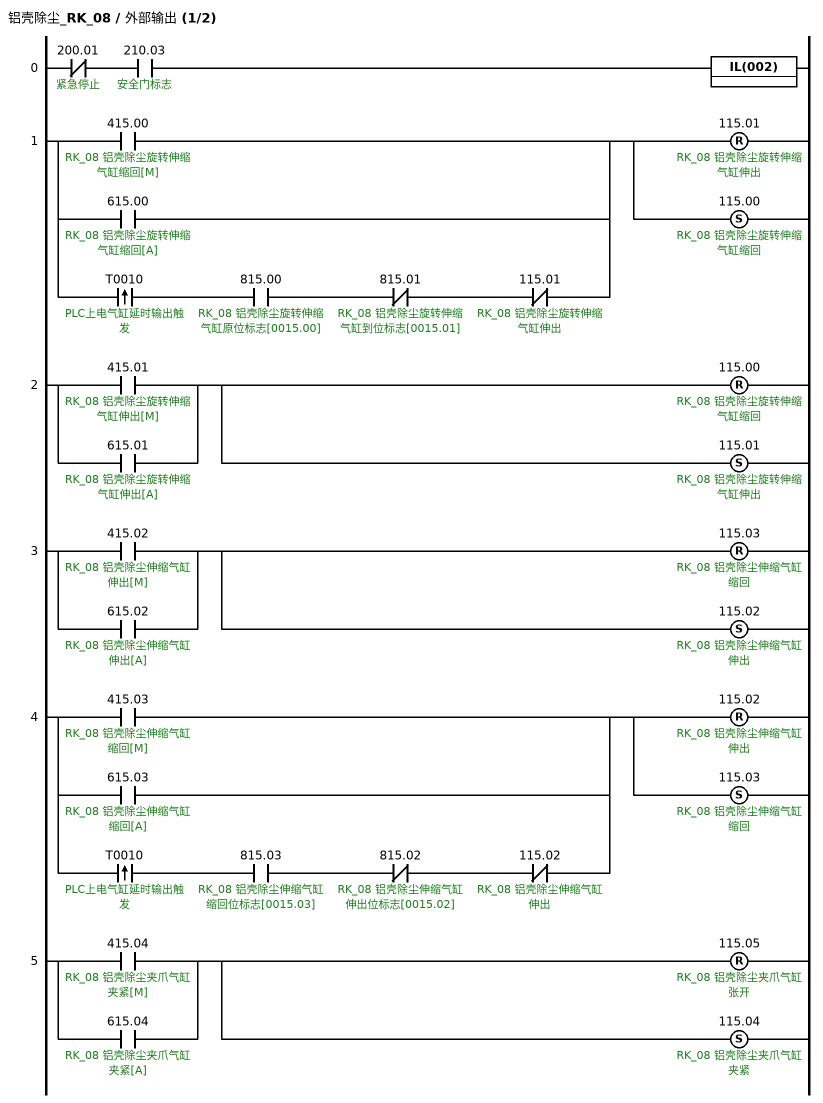
; rung 0
LDNOT 200.01  ; 紧急停止
AND 210.03  ; 安全门标志
IL(002)
; rung 1
LD 415.00  ; RK_08 铝壳除尘旋转伸缩气缸缩回[M]
OR 615.00  ; RK_08 铝壳除尘旋转伸缩气缸缩回[A]
@LD T0010  ; PLC上电气缸延时输出触发
AND 815.00  ; RK_08 铝壳除尘旋转伸缩气缸原位标志[0015.00]
ANDNOT 815.01  ; RK_08 铝壳除尘旋转伸缩气缸到位标志[0015.01]
ANDNOT 115.01  ; RK_08 铝壳除尘旋转伸缩气缸伸出
ORLD
RSET 115.01  ; RK_08 铝壳除尘旋转伸缩气缸伸出
SET 115.00  ; RK_08 铝壳除尘旋转伸缩气缸缩回
; rung 2
LD 415.01  ; RK_08 铝壳除尘旋转伸缩气缸伸出[M]
OR 615.01  ; RK_08 铝壳除尘旋转伸缩气缸伸出[A]
RSET 115.00  ; RK_08 铝壳除尘旋转伸缩气缸缩回
SET 115.01  ; RK_08 铝壳除尘旋转伸缩气缸伸出
; rung 3
LD 415.02  ; RK_08 铝壳除尘伸缩气缸伸出[M]
OR 615.02  ; RK_08 铝壳除尘伸缩气缸伸出[A]
RSET 115.03  ; RK_08 铝壳除尘伸缩气缸缩回
SET 115.02  ; RK_08 铝壳除尘伸缩气缸伸出
; rung 4
LD 415.03  ; RK_08 铝壳除尘伸缩气缸缩回[M]
OR 615.03  ; RK_08 铝壳除尘伸缩气缸缩回[A]
@LD T0010  ; PLC上电气缸延时输出触发
AND 815.03  ; RK_08 铝壳除尘伸缩气缸缩回位标志[0015.03]
ANDNOT 815.02  ; RK_08 铝壳除尘伸缩气缸伸出位标志[0015.02]
ANDNOT 115.02  ; RK_08 铝壳除尘伸缩气缸伸出
ORLD
RSET 115.02  ; RK_08 铝壳除尘伸缩气缸伸出
SET 115.03  ; RK_08 铝壳除尘伸缩气缸缩回
; rung 5
LD 415.04  ; RK_08 铝壳除尘夹爪气缸夹紧[M]
OR 615.04  ; RK_08 铝壳除尘夹爪气缸夹紧[A]
RSET 115.05  ; RK_08 铝壳除尘夹爪气缸张开
SET 115.04  ; RK_08 铝壳除尘夹爪气缸夹紧

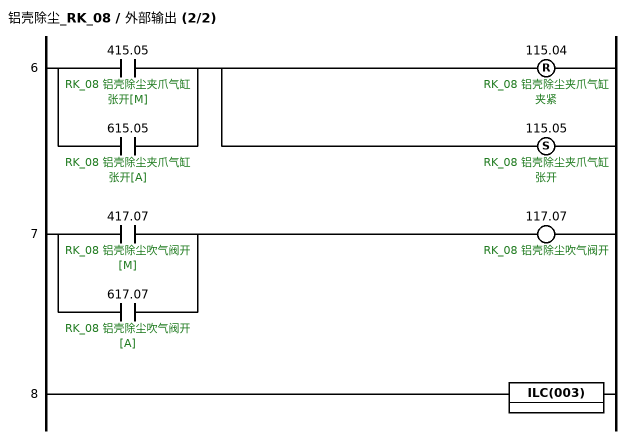
; rung 6
LD 415.05  ; RK_08 铝壳除尘夹爪气缸张开[M]
OR 615.05  ; RK_08 铝壳除尘夹爪气缸张开[A]
RSET 115.04  ; RK_08 铝壳除尘夹爪气缸夹紧
SET 115.05  ; RK_08 铝壳除尘夹爪气缸张开
; rung 7
LD 417.07  ; RK_08 铝壳除尘吹气阀开[M]
OR 617.07  ; RK_08 铝壳除尘吹气阀开[A]
OUT 117.07  ; RK_08 铝壳除尘吹气阀开
; rung 8
ILC(003)

### Section END
; rung 0
END(001)

## Program Hipot检测_RK_09 (cyclic task 9)

### Section Main_1Hipot检测

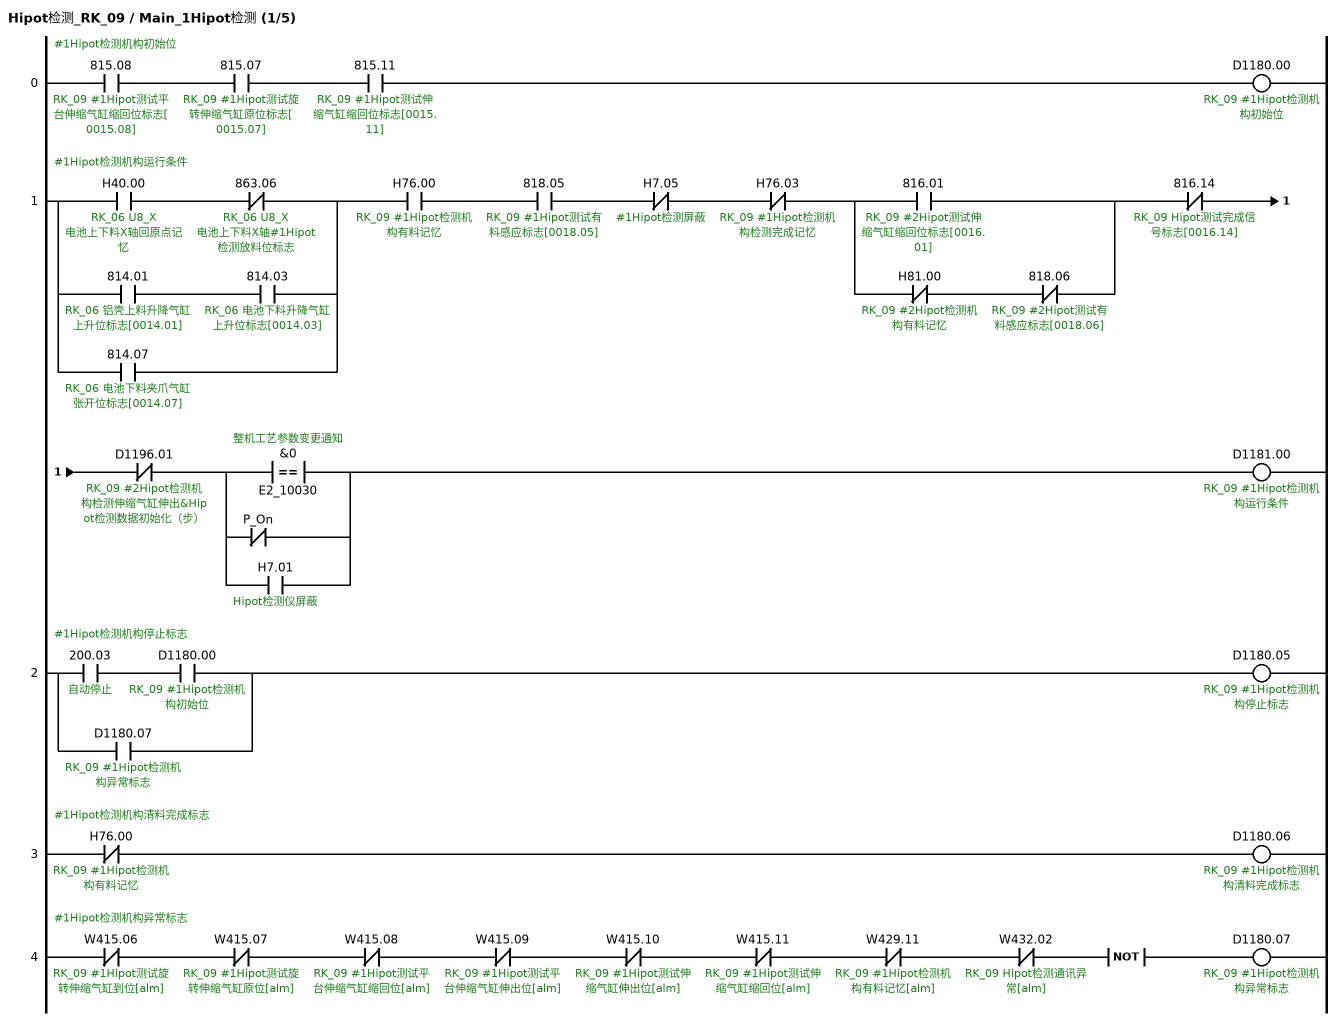
; rung 0: #1Hipot检测机构初始位
LD 815.08  ; RK_09 #1Hipot测试平台伸缩气缸缩回位标志[0015.08]
AND 815.07  ; RK_09 #1Hipot测试旋转伸缩气缸原位标志[0015.07]
AND 815.11  ; RK_09 #1Hipot测试伸缩气缸缩回位标志[0015.11]
OUT D1180.00  ; RK_09 #1Hipot检测机构初始位
; rung 1: #1Hipot检测机构运行条件
LD H40.00  ; RK_06 U8_X 电池上下料X轴回原点记忆
ANDNOT 863.06  ; RK_06 U8_X 电池上下料X轴#1Hipot检测放料位标志
LD 814.01  ; RK_06 铝壳上料升降气缸上升位标志[0014.01]
AND 814.03  ; RK_06 电池下料升降气缸上升位标志[0014.03]
ORLD
OR 814.07  ; RK_06 电池下料夹爪气缸张开位标志[0014.07]
AND H76.00  ; RK_09 #1Hipot检测机构有料记忆
AND 818.05  ; RK_09 #1Hipot测试有料感应标志[0018.05]
ANDNOT H7.05  ; #1Hipot检测屏蔽
ANDNOT H76.03  ; RK_09 #1Hipot检测机构检测完成记忆
LD 816.01  ; RK_09 #2Hipot测试伸缩气缸缩回位标志[0016.01]
LDNOT H81.00  ; RK_09 #2Hipot检测机构有料记忆
ANDNOT 818.06  ; RK_09 #2Hipot测试有料感应标志[0018.06]
ORLD
ANDLD
ANDNOT 816.14  ; RK_09 Hipot测试完成信号标志[0016.14]
ANDNOT D1196.01  ; RK_09 #2Hipot检测机构检测伸缩气缸伸出&Hipot检测数据初始化（步）
LD=(300) &0 E2_10030  ; 整机工艺参数变更通知
ORNOT P_On
OR H7.01  ; Hipot检测仪屏蔽
ANDLD
OUT D1181.00  ; RK_09 #1Hipot检测机构运行条件
; rung 2: #1Hipot检测机构停止标志
LD 200.03  ; 自动停止
AND D1180.00  ; RK_09 #1Hipot检测机构初始位
OR D1180.07  ; RK_09 #1Hipot检测机构异常标志
OUT D1180.05  ; RK_09 #1Hipot检测机构停止标志
; rung 3: #1Hipot检测机构清料完成标志
LDNOT H76.00  ; RK_09 #1Hipot检测机构有料记忆
OUT D1180.06  ; RK_09 #1Hipot检测机构清料完成标志
; rung 4: #1Hipot检测机构异常标志
LDNOT W415.06  ; RK_09 #1Hipot测试旋转伸缩气缸到位[alm]
ANDNOT W415.07  ; RK_09 #1Hipot测试旋转伸缩气缸原位[alm]
ANDNOT W415.08  ; RK_09 #1Hipot测试平台伸缩气缸缩回位[alm]
ANDNOT W415.09  ; RK_09 #1Hipot测试平台伸缩气缸伸出位[alm]
ANDNOT W415.10  ; RK_09 #1Hipot测试伸缩气缸伸出位[alm]
ANDNOT W415.11  ; RK_09 #1Hipot测试伸缩气缸缩回位[alm]
ANDNOT W429.11  ; RK_09 #1Hipot检测机构有料记忆[alm]
ANDNOT W432.02  ; RK_09 Hipot检测通讯异常[alm]
NOT(520)
OUT D1180.07  ; RK_09 #1Hipot检测机构异常标志

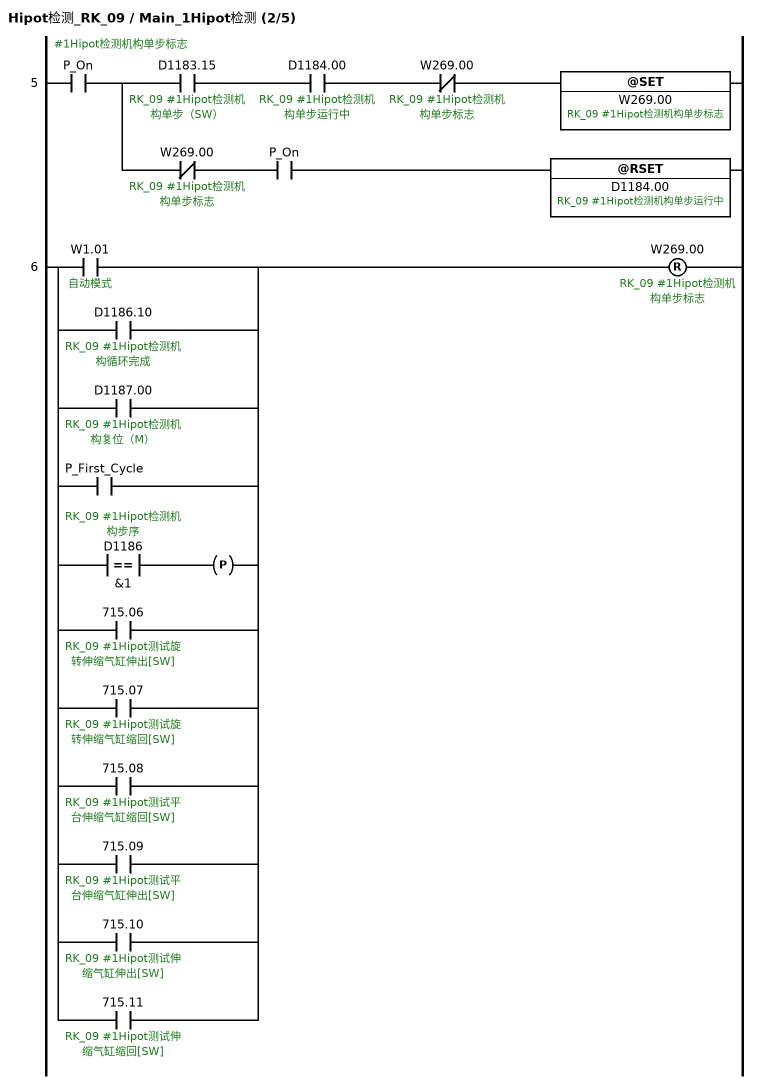
; rung 5: #1Hipot检测机构单步标志
LD P_On
OUT TR0
AND D1183.15  ; RK_09 #1Hipot检测机构单步（SW）
AND D1184.00  ; RK_09 #1Hipot检测机构单步运行中
ANDNOT W269.00  ; RK_09 #1Hipot检测机构单步标志
@SET W269.00  ; RK_09 #1Hipot检测机构单步标志
LD TR0
ANDNOT W269.00  ; RK_09 #1Hipot检测机构单步标志
AND P_On
@RSET D1184.00  ; RK_09 #1Hipot检测机构单步运行中
; rung 6
LD W1.01  ; 自动模式
OR D1186.10  ; RK_09 #1Hipot检测机构循环完成
OR D1187.00  ; RK_09 #1Hipot检测机构复位（M）
OR P_First_Cycle
LD=(300) D1186 &1  ; RK_09 #1Hipot检测机构步序
UP(521)
ORLD
OR 715.06  ; RK_09 #1Hipot测试旋转伸缩气缸伸出[SW]
OR 715.07  ; RK_09 #1Hipot测试旋转伸缩气缸缩回[SW]
OR 715.08  ; RK_09 #1Hipot测试平台伸缩气缸缩回[SW]
OR 715.09  ; RK_09 #1Hipot测试平台伸缩气缸伸出[SW]
OR 715.10  ; RK_09 #1Hipot测试伸缩气缸伸出[SW]
OR 715.11  ; RK_09 #1Hipot测试伸缩气缸缩回[SW]
RSET W269.00  ; RK_09 #1Hipot检测机构单步标志

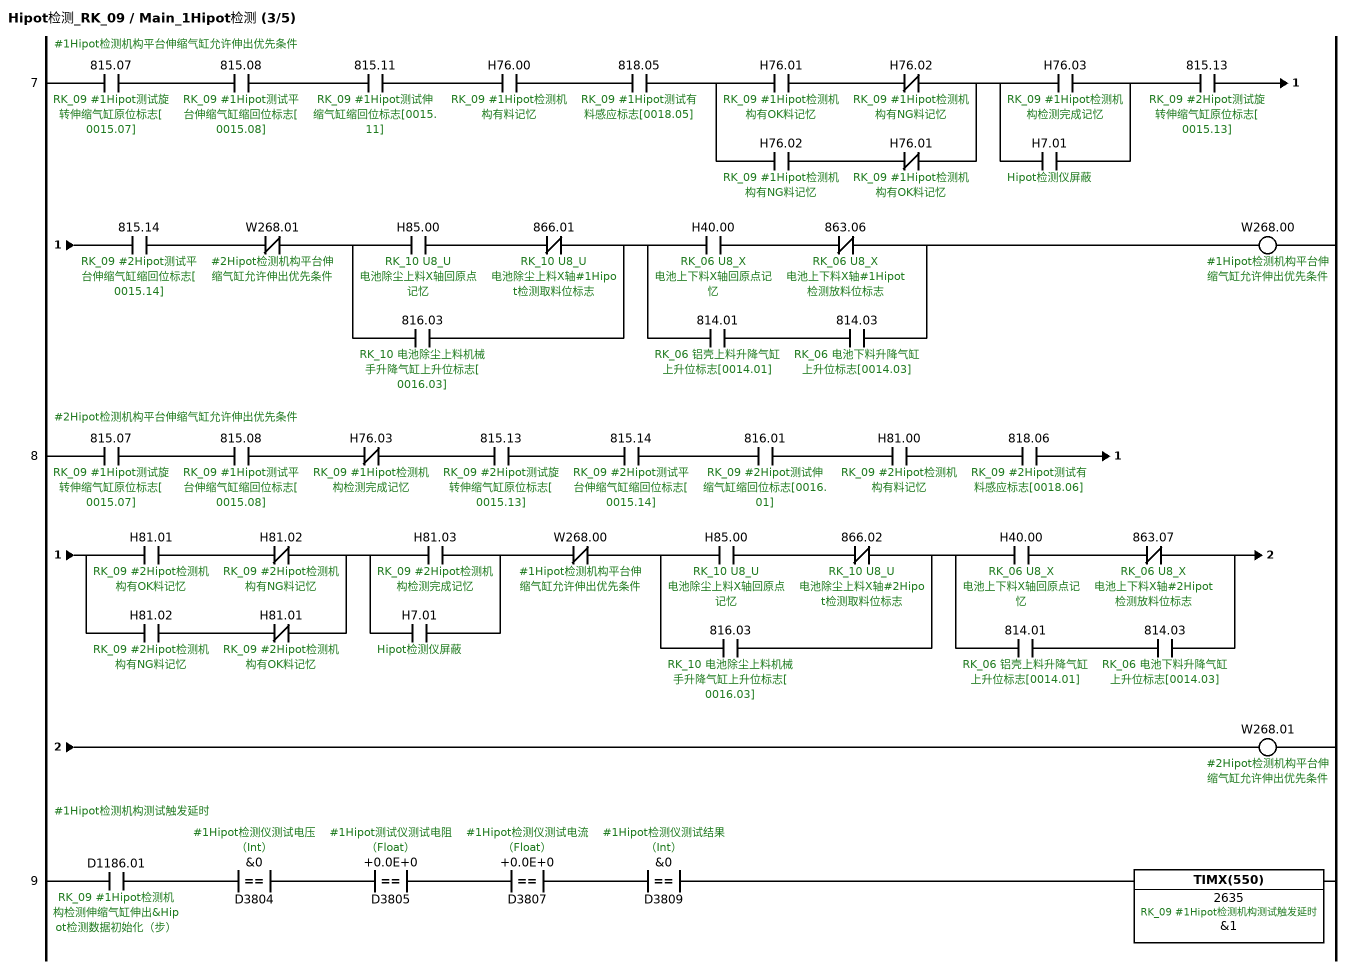
; rung 7: #1Hipot检测机构平台伸缩气缸允许伸出优先条件
LD 815.07  ; RK_09 #1Hipot测试旋转伸缩气缸原位标志[0015.07]
AND 815.08  ; RK_09 #1Hipot测试平台伸缩气缸缩回位标志[0015.08]
AND 815.11  ; RK_09 #1Hipot测试伸缩气缸缩回位标志[0015.11]
AND H76.00  ; RK_09 #1Hipot检测机构有料记忆
AND 818.05  ; RK_09 #1Hipot测试有料感应标志[0018.05]
LD H76.01  ; RK_09 #1Hipot检测机构有OK料记忆
ANDNOT H76.02  ; RK_09 #1Hipot检测机构有NG料记忆
LD H76.02  ; RK_09 #1Hipot检测机构有NG料记忆
ANDNOT H76.01  ; RK_09 #1Hipot检测机构有OK料记忆
ORLD
ANDLD
LD H76.03  ; RK_09 #1Hipot检测机构检测完成记忆
OR H7.01  ; Hipot检测仪屏蔽
ANDLD
AND 815.13  ; RK_09 #2Hipot测试旋转伸缩气缸原位标志[0015.13]
AND 815.14  ; RK_09 #2Hipot测试平台伸缩气缸缩回位标志[0015.14]
ANDNOT W268.01  ; #2Hipot检测机构平台伸缩气缸允许伸出优先条件
LD H85.00  ; RK_10 U8_U 电池除尘上料X轴回原点记忆
ANDNOT 866.01  ; RK_10 U8_U 电池除尘上料X轴#1Hipot检测取料位标志
OR 816.03  ; RK_10 电池除尘上料机械手升降气缸上升位标志[0016.03]
ANDLD
LD H40.00  ; RK_06 U8_X 电池上下料X轴回原点记忆
ANDNOT 863.06  ; RK_06 U8_X 电池上下料X轴#1Hipot检测放料位标志
LD 814.01  ; RK_06 铝壳上料升降气缸上升位标志[0014.01]
AND 814.03  ; RK_06 电池下料升降气缸上升位标志[0014.03]
ORLD
ANDLD
OUT W268.00  ; #1Hipot检测机构平台伸缩气缸允许伸出优先条件
; rung 8: #2Hipot检测机构平台伸缩气缸允许伸出优先条件
LD 815.07  ; RK_09 #1Hipot测试旋转伸缩气缸原位标志[0015.07]
AND 815.08  ; RK_09 #1Hipot测试平台伸缩气缸缩回位标志[0015.08]
ANDNOT H76.03  ; RK_09 #1Hipot检测机构检测完成记忆
AND 815.13  ; RK_09 #2Hipot测试旋转伸缩气缸原位标志[0015.13]
AND 815.14  ; RK_09 #2Hipot测试平台伸缩气缸缩回位标志[0015.14]
AND 816.01  ; RK_09 #2Hipot测试伸缩气缸缩回位标志[0016.01]
AND H81.00  ; RK_09 #2Hipot检测机构有料记忆
AND 818.06  ; RK_09 #2Hipot测试有料感应标志[0018.06]
LD H81.01  ; RK_09 #2Hipot检测机构有OK料记忆
ANDNOT H81.02  ; RK_09 #2Hipot检测机构有NG料记忆
LD H81.02  ; RK_09 #2Hipot检测机构有NG料记忆
ANDNOT H81.01  ; RK_09 #2Hipot检测机构有OK料记忆
ORLD
ANDLD
LD H81.03  ; RK_09 #2Hipot检测机构检测完成记忆
OR H7.01  ; Hipot检测仪屏蔽
ANDLD
ANDNOT W268.00  ; #1Hipot检测机构平台伸缩气缸允许伸出优先条件
LD H85.00  ; RK_10 U8_U 电池除尘上料X轴回原点记忆
ANDNOT 866.02  ; RK_10 U8_U 电池除尘上料X轴#2Hipot检测取料位标志
OR 816.03  ; RK_10 电池除尘上料机械手升降气缸上升位标志[0016.03]
ANDLD
LD H40.00  ; RK_06 U8_X 电池上下料X轴回原点记忆
ANDNOT 863.07  ; RK_06 U8_X 电池上下料X轴#2Hipot检测放料位标志
LD 814.01  ; RK_06 铝壳上料升降气缸上升位标志[0014.01]
AND 814.03  ; RK_06 电池下料升降气缸上升位标志[0014.03]
ORLD
ANDLD
OUT W268.01  ; #2Hipot检测机构平台伸缩气缸允许伸出优先条件
; rung 9: #1Hipot检测机构测试触发延时
LD D1186.01  ; RK_09 #1Hipot检测机构检测伸缩气缸伸出&Hipot检测数据初始化（步）
AND=(300) &0 D3804  ; #1Hipot检测仪测试电压（Int）
AND=F(329) +0.0E+0 D3805  ; #1Hipot测试仪测试电阻（Float）
AND=F(329) +0.0E+0 D3807  ; #1Hipot检测仪测试电流（Float）
AND=(300) &0 D3809  ; #1Hipot检测仪测试结果（Int）
TIMX(550) 2635 &1  ; RK_09 #1Hipot检测机构测试触发延时

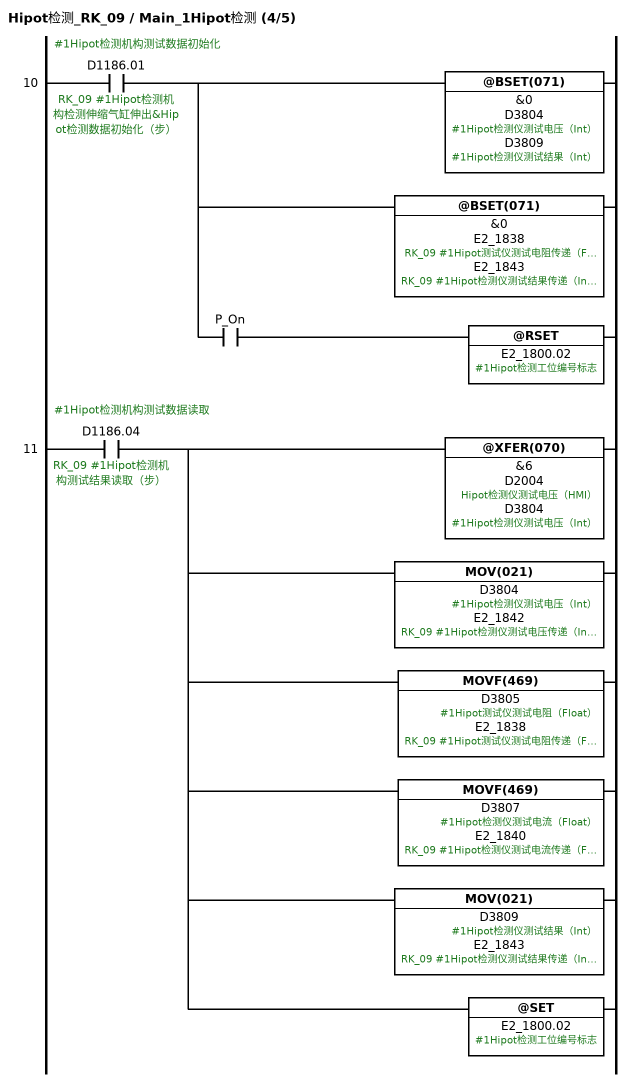
; rung 10: #1Hipot检测机构测试数据初始化
LD D1186.01  ; RK_09 #1Hipot检测机构检测伸缩气缸伸出&Hipot检测数据初始化（步）
@BSET(071) &0 D3804 D3809  ; #1Hipot检测仪测试电压（Int）, #1Hipot检测仪测试结果（Int）
@BSET(071) &0 E2_1838 E2_1843  ; RK_09 #1Hipot测试仪测试电阻传递（Float）, RK_09 #1Hipot检测仪测试结果传递（Int）
AND P_On
@RSET E2_1800.02  ; #1Hipot检测工位编号标志
; rung 11: #1Hipot检测机构测试数据读取
LD D1186.04  ; RK_09 #1Hipot检测机构测试结果读取（步）
@XFER(070) &6 D2004 D3804  ; Hipot检测仪测试电压（HMI）, #1Hipot检测仪测试电压（Int）
MOV(021) D3804 E2_1842  ; #1Hipot检测仪测试电压（Int）, RK_09 #1Hipot检测仪测试电压传递（Int）
MOVF(469) D3805 E2_1838  ; #1Hipot测试仪测试电阻（Float）, RK_09 #1Hipot测试仪测试电阻传递（Float）
MOVF(469) D3807 E2_1840  ; #1Hipot检测仪测试电流（Float）, RK_09 #1Hipot检测仪测试电流传递（Float）
MOV(021) D3809 E2_1843  ; #1Hipot检测仪测试结果（Int）, RK_09 #1Hipot检测仪测试结果传递（Int）
@SET E2_1800.02  ; #1Hipot检测工位编号标志

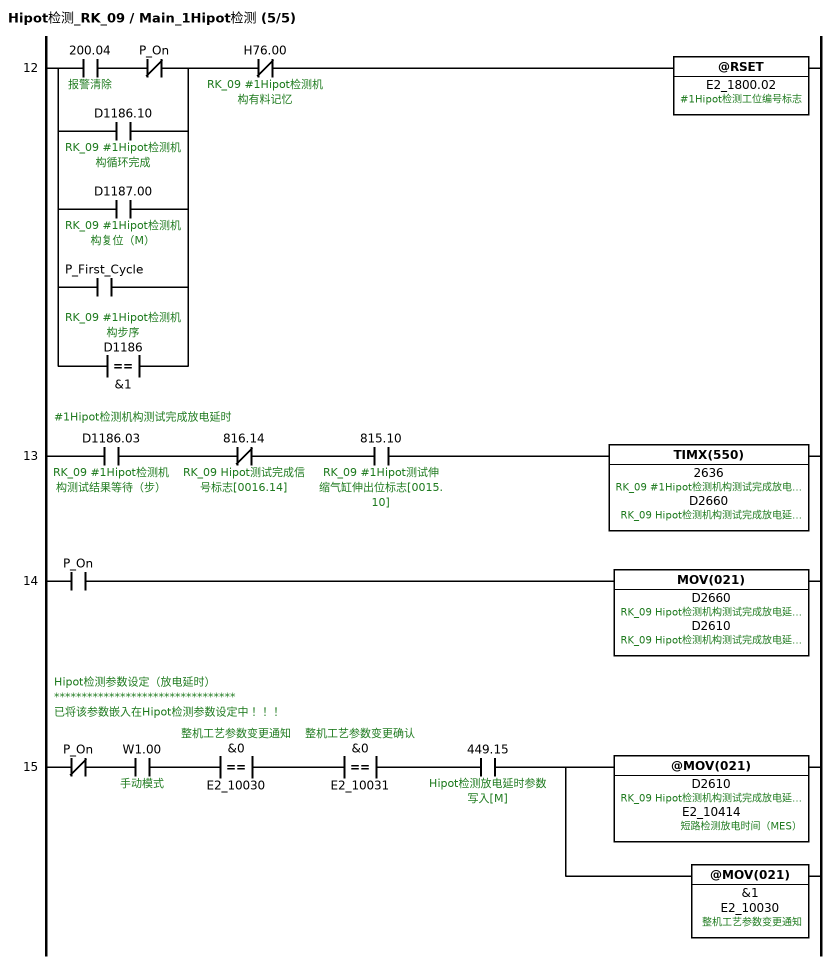
; rung 12
LD 200.04  ; 报警清除
ANDNOT P_On
OR D1186.10  ; RK_09 #1Hipot检测机构循环完成
OR D1187.00  ; RK_09 #1Hipot检测机构复位（M）
OR P_First_Cycle
OR=(300) D1186 &1  ; RK_09 #1Hipot检测机构步序
ANDNOT H76.00  ; RK_09 #1Hipot检测机构有料记忆
@RSET E2_1800.02  ; #1Hipot检测工位编号标志
; rung 13: #1Hipot检测机构测试完成放电延时
LD D1186.03  ; RK_09 #1Hipot检测机构测试结果等待（步）
ANDNOT 816.14  ; RK_09 Hipot测试完成信号标志[0016.14]
AND 815.10  ; RK_09 #1Hipot测试伸缩气缸伸出位标志[0015.10]
TIMX(550) 2636 D2660  ; RK_09 Hipot检测机构测试完成放电延时设定, RK_09 #1Hipot检测机构测试完成放电延时
; rung 14
LD P_On
MOV(021) D2660 D2610  ; RK_09 Hipot检测机构测试完成放电延时设定, RK_09 Hipot检测机构测试完成放电延时参数设定
; rung 15: Hipot检测参数设定（放电延时） / ********************************* / 已将该参数嵌入在Hipot检测参数设定中！！！
LDNOT P_On
AND W1.00  ; 手动模式
AND=(300) &0 E2_10030  ; 整机工艺参数变更通知
AND=(300) &0 E2_10031  ; 整机工艺参数变更确认
AND 449.15  ; Hipot检测放电延时参数写入[M]
@MOV(021) D2610 E2_10414  ; RK_09 Hipot检测机构测试完成放电延时参数设定, 短路检测放电时间（MES）
@MOV(021) &1 E2_10030  ; 整机工艺参数变更通知

### Section Main_2Hipot检测

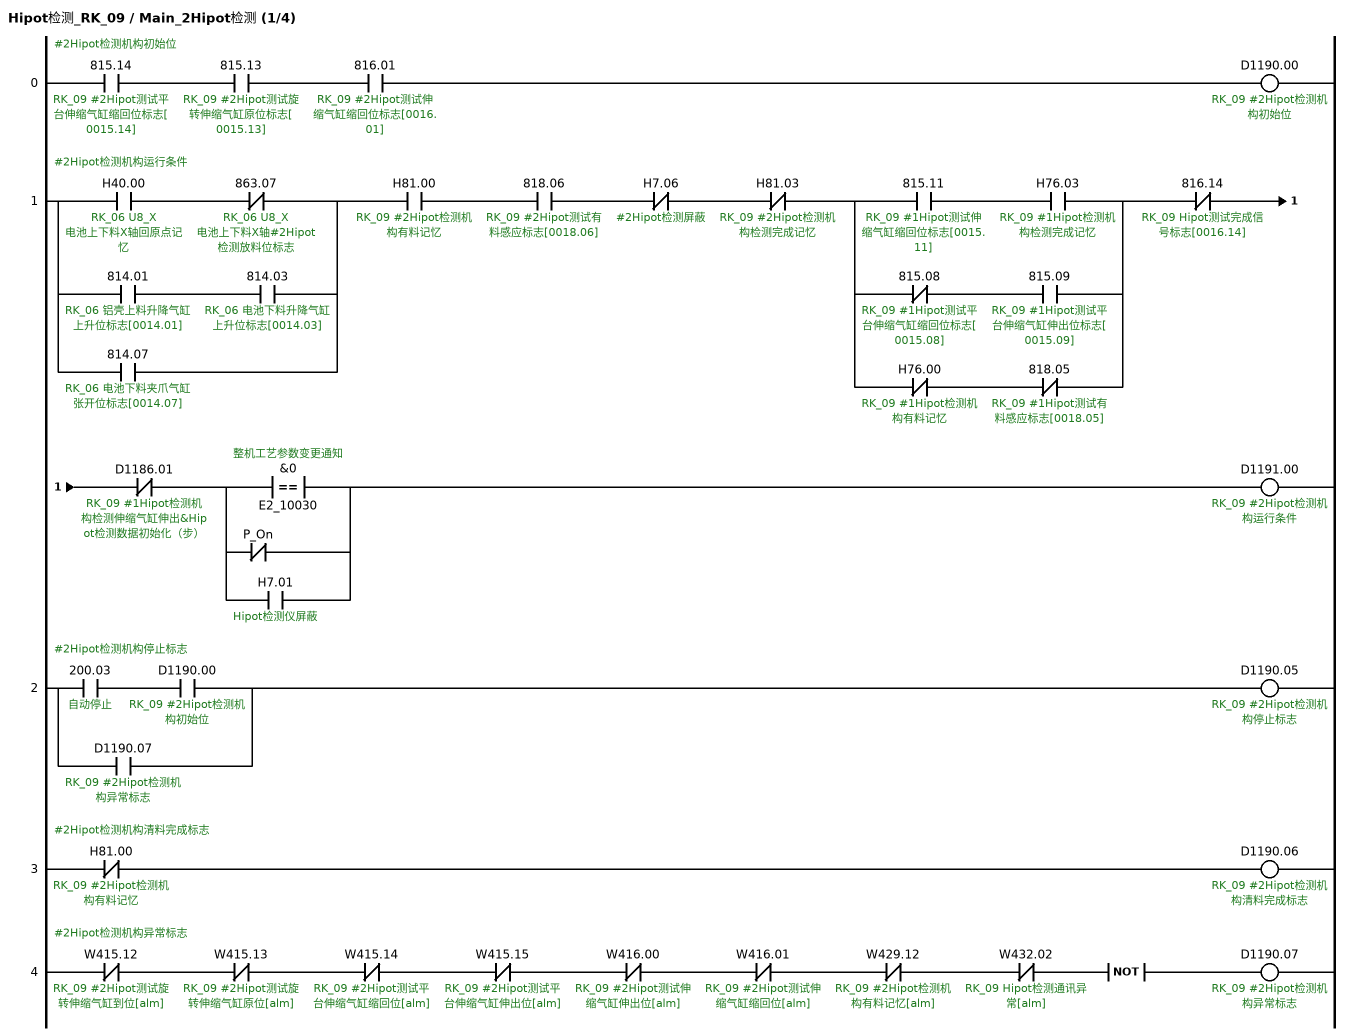
; rung 0: #2Hipot检测机构初始位
LD 815.14  ; RK_09 #2Hipot测试平台伸缩气缸缩回位标志[0015.14]
AND 815.13  ; RK_09 #2Hipot测试旋转伸缩气缸原位标志[0015.13]
AND 816.01  ; RK_09 #2Hipot测试伸缩气缸缩回位标志[0016.01]
OUT D1190.00  ; RK_09 #2Hipot检测机构初始位
; rung 1: #2Hipot检测机构运行条件
LD H40.00  ; RK_06 U8_X 电池上下料X轴回原点记忆
ANDNOT 863.07  ; RK_06 U8_X 电池上下料X轴#2Hipot检测放料位标志
LD 814.01  ; RK_06 铝壳上料升降气缸上升位标志[0014.01]
AND 814.03  ; RK_06 电池下料升降气缸上升位标志[0014.03]
ORLD
OR 814.07  ; RK_06 电池下料夹爪气缸张开位标志[0014.07]
AND H81.00  ; RK_09 #2Hipot检测机构有料记忆
AND 818.06  ; RK_09 #2Hipot测试有料感应标志[0018.06]
ANDNOT H7.06  ; #2Hipot检测屏蔽
ANDNOT H81.03  ; RK_09 #2Hipot检测机构检测完成记忆
LD 815.11  ; RK_09 #1Hipot测试伸缩气缸缩回位标志[0015.11]
AND H76.03  ; RK_09 #1Hipot检测机构检测完成记忆
LDNOT 815.08  ; RK_09 #1Hipot测试平台伸缩气缸缩回位标志[0015.08]
AND 815.09  ; RK_09 #1Hipot测试平台伸缩气缸伸出位标志[0015.09]
ORLD
LDNOT H76.00  ; RK_09 #1Hipot检测机构有料记忆
ANDNOT 818.05  ; RK_09 #1Hipot测试有料感应标志[0018.05]
ORLD
ANDLD
ANDNOT 816.14  ; RK_09 Hipot测试完成信号标志[0016.14]
ANDNOT D1186.01  ; RK_09 #1Hipot检测机构检测伸缩气缸伸出&Hipot检测数据初始化（步）
LD=(300) &0 E2_10030  ; 整机工艺参数变更通知
ORNOT P_On
OR H7.01  ; Hipot检测仪屏蔽
ANDLD
OUT D1191.00  ; RK_09 #2Hipot检测机构运行条件
; rung 2: #2Hipot检测机构停止标志
LD 200.03  ; 自动停止
AND D1190.00  ; RK_09 #2Hipot检测机构初始位
OR D1190.07  ; RK_09 #2Hipot检测机构异常标志
OUT D1190.05  ; RK_09 #2Hipot检测机构停止标志
; rung 3: #2Hipot检测机构清料完成标志
LDNOT H81.00  ; RK_09 #2Hipot检测机构有料记忆
OUT D1190.06  ; RK_09 #2Hipot检测机构清料完成标志
; rung 4: #2Hipot检测机构异常标志
LDNOT W415.12  ; RK_09 #2Hipot测试旋转伸缩气缸到位[alm]
ANDNOT W415.13  ; RK_09 #2Hipot测试旋转伸缩气缸原位[alm]
ANDNOT W415.14  ; RK_09 #2Hipot测试平台伸缩气缸缩回位[alm]
ANDNOT W415.15  ; RK_09 #2Hipot测试平台伸缩气缸伸出位[alm]
ANDNOT W416.00  ; RK_09 #2Hipot测试伸缩气缸伸出位[alm]
ANDNOT W416.01  ; RK_09 #2Hipot测试伸缩气缸缩回位[alm]
ANDNOT W429.12  ; RK_09 #2Hipot检测机构有料记忆[alm]
ANDNOT W432.02  ; RK_09 Hipot检测通讯异常[alm]
NOT(520)
OUT D1190.07  ; RK_09 #2Hipot检测机构异常标志

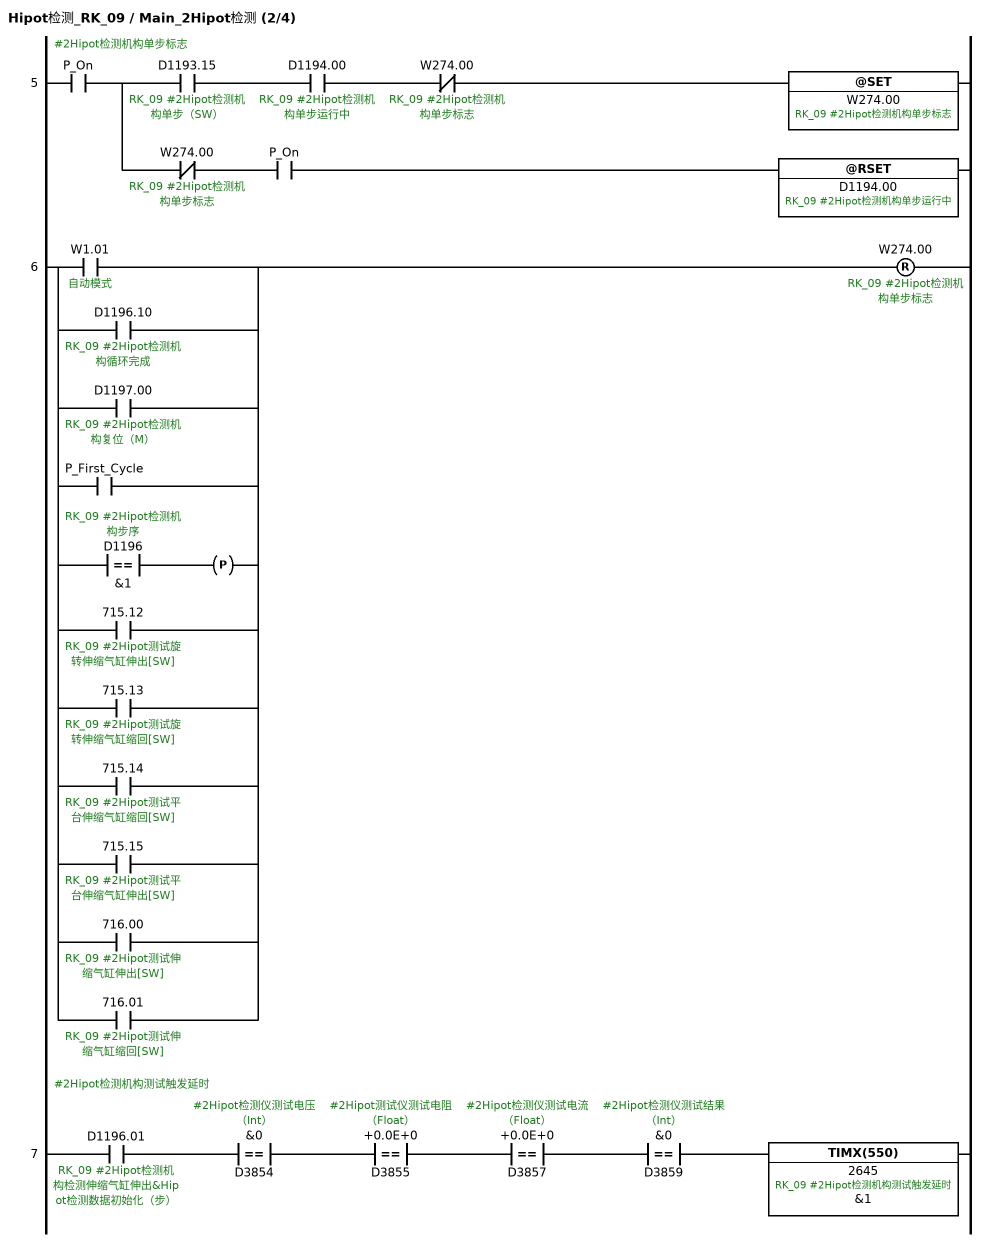
; rung 5: #2Hipot检测机构单步标志
LD P_On
OUT TR0
AND D1193.15  ; RK_09 #2Hipot检测机构单步（SW）
AND D1194.00  ; RK_09 #2Hipot检测机构单步运行中
ANDNOT W274.00  ; RK_09 #2Hipot检测机构单步标志
@SET W274.00  ; RK_09 #2Hipot检测机构单步标志
LD TR0
ANDNOT W274.00  ; RK_09 #2Hipot检测机构单步标志
AND P_On
@RSET D1194.00  ; RK_09 #2Hipot检测机构单步运行中
; rung 6
LD W1.01  ; 自动模式
OR D1196.10  ; RK_09 #2Hipot检测机构循环完成
OR D1197.00  ; RK_09 #2Hipot检测机构复位（M）
OR P_First_Cycle
LD=(300) D1196 &1  ; RK_09 #2Hipot检测机构步序
UP(521)
ORLD
OR 715.12  ; RK_09 #2Hipot测试旋转伸缩气缸伸出[SW]
OR 715.13  ; RK_09 #2Hipot测试旋转伸缩气缸缩回[SW]
OR 715.14  ; RK_09 #2Hipot测试平台伸缩气缸缩回[SW]
OR 715.15  ; RK_09 #2Hipot测试平台伸缩气缸伸出[SW]
OR 716.00  ; RK_09 #2Hipot测试伸缩气缸伸出[SW]
OR 716.01  ; RK_09 #2Hipot测试伸缩气缸缩回[SW]
RSET W274.00  ; RK_09 #2Hipot检测机构单步标志
; rung 7: #2Hipot检测机构测试触发延时
LD D1196.01  ; RK_09 #2Hipot检测机构检测伸缩气缸伸出&Hipot检测数据初始化（步）
AND=(300) &0 D3854  ; #2Hipot检测仪测试电压（Int）
AND=F(329) +0.0E+0 D3855  ; #2Hipot测试仪测试电阻（Float）
AND=F(329) +0.0E+0 D3857  ; #2Hipot检测仪测试电流（Float）
AND=(300) &0 D3859  ; #2Hipot检测仪测试结果（Int）
TIMX(550) 2645 &1  ; RK_09 #2Hipot检测机构测试触发延时

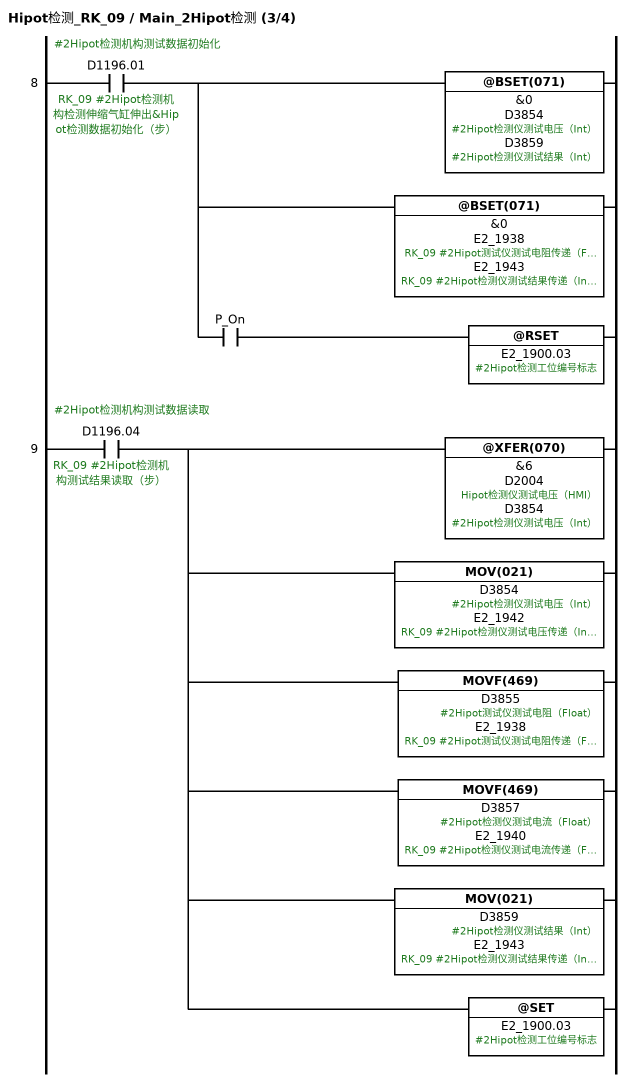
; rung 8: #2Hipot检测机构测试数据初始化
LD D1196.01  ; RK_09 #2Hipot检测机构检测伸缩气缸伸出&Hipot检测数据初始化（步）
@BSET(071) &0 D3854 D3859  ; #2Hipot检测仪测试电压（Int）, #2Hipot检测仪测试结果（Int）
@BSET(071) &0 E2_1938 E2_1943  ; RK_09 #2Hipot测试仪测试电阻传递（Float）, RK_09 #2Hipot检测仪测试结果传递（Int）
AND P_On
@RSET E2_1900.03  ; #2Hipot检测工位编号标志
; rung 9: #2Hipot检测机构测试数据读取
LD D1196.04  ; RK_09 #2Hipot检测机构测试结果读取（步）
@XFER(070) &6 D2004 D3854  ; Hipot检测仪测试电压（HMI）, #2Hipot检测仪测试电压（Int）
MOV(021) D3854 E2_1942  ; #2Hipot检测仪测试电压（Int）, RK_09 #2Hipot检测仪测试电压传递（Int）
MOVF(469) D3855 E2_1938  ; #2Hipot测试仪测试电阻（Float）, RK_09 #2Hipot测试仪测试电阻传递（Float）
MOVF(469) D3857 E2_1940  ; #2Hipot检测仪测试电流（Float）, RK_09 #2Hipot检测仪测试电流传递（Float）
MOV(021) D3859 E2_1943  ; #2Hipot检测仪测试结果（Int）, RK_09 #2Hipot检测仪测试结果传递（Int）
@SET E2_1900.03  ; #2Hipot检测工位编号标志

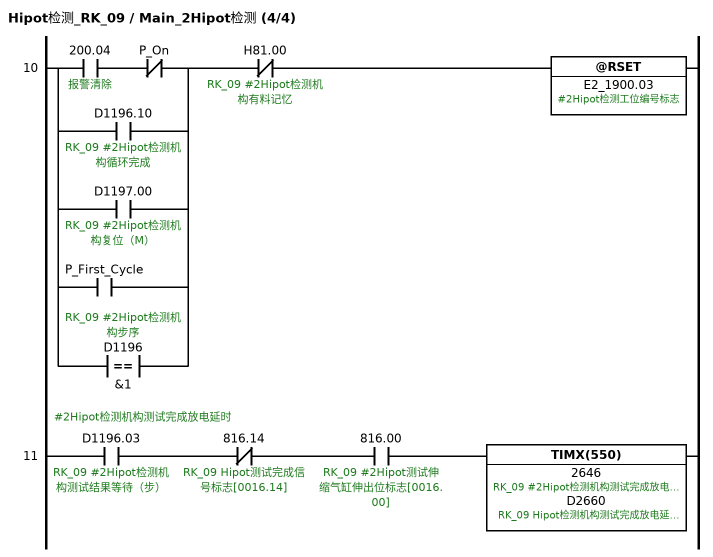
; rung 10
LD 200.04  ; 报警清除
ANDNOT P_On
OR D1196.10  ; RK_09 #2Hipot检测机构循环完成
OR D1197.00  ; RK_09 #2Hipot检测机构复位（M）
OR P_First_Cycle
OR=(300) D1196 &1  ; RK_09 #2Hipot检测机构步序
ANDNOT H81.00  ; RK_09 #2Hipot检测机构有料记忆
@RSET E2_1900.03  ; #2Hipot检测工位编号标志
; rung 11: #2Hipot检测机构测试完成放电延时
LD D1196.03  ; RK_09 #2Hipot检测机构测试结果等待（步）
ANDNOT 816.14  ; RK_09 Hipot测试完成信号标志[0016.14]
AND 816.00  ; RK_09 #2Hipot测试伸缩气缸伸出位标志[0016.00]
TIMX(550) 2646 D2660  ; RK_09 Hipot检测机构测试完成放电延时设定, RK_09 #2Hipot检测机构测试完成放电延时

### Section 手动_1Hipot检测

